KUKA KRL program: MyProgram_014().src

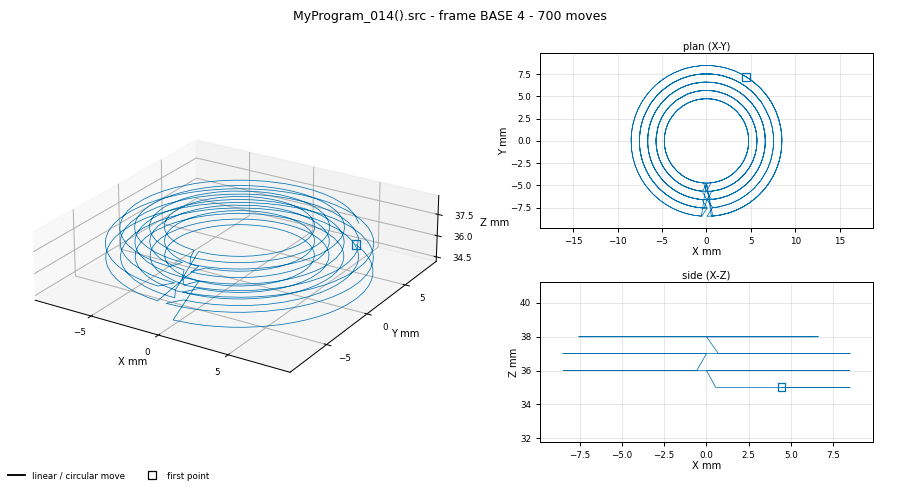
[picture p0: tool path of MyProgram_014().src in frame BASE 4, 700 of 700 moves have a stored position in this frame; points joined in program order, loops and branches not executed]
&ACCESS RVP
&REL 1
&PARAM TEMPLATE = C:\KRC\Roboter\Template\vorgabe
&PARAM EDITMASK = *
DEF MyProgram_014()
; ---- Setting reference (Base) ----
$BASE = BASE_DATA[4]

; --------------------------
; ---- Setting tool (TCP) ----
$TOOL = TOOL_DATA[3]
; --------------------------

$VEL.CP = VEL_APROX_PRINT
Startdeposition()
$VEL.CP = VEL_PRINT
LIN {X 4.4354,Y 7.2394,Z 35,A -2.2302,B 0,C 0,E1 0.1598,E2 90.0725} C_DIS
LIN {X 5.4049,Y 6.549,Z 35,A -2.2236,B 0,C 0,E1 0.1598,E2 90.0723} C_DIS
LIN {X 6.1861,Y 5.8118,Z 35,A -2.2262,B 0,C 0,E1 0.1598,E2 90.0723} C_DIS
LIN {X 6.7419,Y 5.1563,Z 35,A -2.2336,B 0,C 0,E1 0.1598,E2 90.0723} C_DIS
LIN {X 7.2287,Y 4.4482,Z 35,A -2.2457,B 0,C 0,E1 0.1598,E2 90.0723} C_DIS
LIN {X 7.6414,Y 3.6945,Z 35,A -2.2626,B 0,C 0,E1 0.1598,E2 90.0723} C_DIS
LIN {X 7.9758,Y 2.9029,Z 35,A -2.2839,B 0,C 0,E1 0.1598,E2 90.0721} C_DIS
LIN {X 8.2282,Y 2.0814,Z 35,A -2.3096,B 0,C 0,E1 0.1598,E2 90.0721} C_DIS
LIN {X 8.3959,Y 1.2387,Z 35,A -2.3393,B 0,C 0,E1 0.1598,E2 90.0721} C_DIS
LIN {X 8.4889,Y 0.1686,Z 35,A -2.3812,B 0,C 0,E1 0.1598,E2 90.0716} C_DIS
LIN {X 8.427,Y -1.0082,Z 35,A -2.4336,B 0,C 0,E1 0.1598,E2 90.0716} C_DIS
LIN {X 8.2841,Y -1.8426,Z 35,A -2.4748,B 0,C 0,E1 0.1598,E2 90.0719} C_DIS
LIN {X 8.0591,Y -2.6586,Z 35,A -2.5179,B 0,C 0,E1 0.1598,E2 90.0719} C_DIS
LIN {X 7.754,Y -3.4482,Z 35,A -2.5628,B 0,C 0,E1 0.1598,E2 90.0719} C_DIS
LIN {X 7.3718,Y -4.2035,Z 35,A -2.6091,B 0,C 0,E1 0.1598,E2 90.0718} C_DIS
LIN {X 6.9163,Y -4.9169,Z 35,A -2.6563,B 0,C 0,E1 0.1598,E2 90.0718} C_DIS
LIN {X 6.3921,Y -5.5815,Z 35,A -2.7039,B 0,C 0,E1 0.1598,E2 90.0718} C_DIS
LIN {X 5.5803,Y -6.3989,Z 35,A -2.7685,B 0,C 0,E1 0.1598,E2 90.0716} C_DIS
LIN {X 4.7589,Y -7.0287,Z 35,A -2.8256,B 0,C 0,E1 0.1598,E2 90.0716} C_DIS
LIN {X 4.0513,Y -7.4589,Z 35,A -2.8699,B 0,C 0,E1 0.1598,E2 90.0716} C_DIS
LIN {X 3.3051,Y -7.8178,Z 35,A -2.9126,B 0,C 0,E1 0.1598,E2 90.0716} C_DIS
LIN {X 2.5274,Y -8.1021,Z 35,A -2.9533,B 0,C 0,E1 0.1598,E2 90.0716} C_DIS
LIN {X 1.7257,Y -8.3091,Z 35,A -2.9915,B 0,C 0,E1 0.1598,E2 90.0716} C_DIS
LIN {X 0.5478,Y -8.4729,Z 35,A -3.0416,B 0,C 0,E1 0.1598,E2 90.0716} C_DIS
LIN {X 0.5478,Y -8.4729,Z 35,A -3.0416,B 0,C 0,E1 0.1598,E2 90.0716} C_DIS
Enddeposition()
LIN {X 0.0007,Y -4.7534,Z 36,A -2.8887,B 0,C 0,E1 0.1598,E2 90.0604} C_DIS
Startdeposition()
$VEL.CP = VEL_PRINT
LIN {X 0.0007,Y -4.7534,Z 36,A -2.8945,B 0,C 0,E1 0.1598,E2 90.0661} C_DIS
LIN {X 0.8257,Y -4.6787,Z 36,A -2.8659,B 0,C 0,E1 0.1598,E2 90.0711} C_DIS
LIN {X 1.4687,Y -4.5179,Z 36,A -2.8361,B 0,C 0,E1 0.1598,E2 90.0717} C_DIS
LIN {X 2.0836,Y -4.2702,Z 36,A -2.803,B 0,C 0,E1 0.1598,E2 90.0718} C_DIS
LIN {X 2.6574,Y -3.9383,Z 36,A -2.7678,B 0,C 0,E1 0.1598,E2 90.0718} C_DIS
LIN {X 3.2997,Y -3.4155,Z 36,A -2.7219,B 0,C 0,E1 0.1598,E2 90.0718} C_DIS
LIN {X 3.7426,Y -2.9228,Z 36,A -2.6846,B 0,C 0,E1 0.1598,E2 90.0718} C_DIS
LIN {X 4.1951,Y -2.2293,Z 36,A -2.6384,B 0,C 0,E1 0.1598,E2 90.0718} C_DIS
LIN {X 4.4644,Y -1.6239,Z 36,A -2.6027,B 0,C 0,E1 0.1598,E2 90.0719} C_DIS
LIN {X 4.6471,Y -0.9868,Z 36,A -2.5689,B 0,C 0,E1 0.1598,E2 90.0719} C_DIS
LIN {X 4.7402,Y -0.3306,Z 36,A -2.5375,B 0,C 0,E1 0.1598,E2 90.0719} C_DIS
LIN {X 4.74,Y 0.3322,Z 36,A -2.5093,B 0,C 0,E1 0.1598,E2 90.0719} C_DIS
LIN {X 4.6474,Y 0.9886,Z 36,A -2.4848,B 0,C 0,E1 0.1598,E2 90.072} C_DIS
LIN {X 4.4647,Y 1.6257,Z 36,A -2.4644,B 0,C 0,E1 0.1598,E2 90.072} C_DIS
LIN {X 4.1961,Y 2.2319,Z 36,A -2.4485,B 0,C 0,E1 0.1598,E2 90.072} C_DIS
LIN {X 3.8438,Y 2.7936,Z 36,A -2.4376,B 0,C 0,E1 0.1598,E2 90.0721} C_DIS
LIN {X 3.4175,Y 3.3013,Z 36,A -2.4318,B 0,C 0,E1 0.1598,E2 90.0721} C_DIS
LIN {X 2.9251,Y 3.7453,Z 36,A -2.4311,B 0,C 0,E1 0.1598,E2 90.0722} C_DIS
LIN {X 2.3754,Y 4.116,Z 36,A -2.4357,B 0,C 0,E1 0.1598,E2 90.0722} C_DIS
LIN {X 1.7795,Y 4.4064,Z 36,A -2.4453,B 0,C 0,E1 0.1598,E2 90.0722} C_DIS
LIN {X 1.149,Y 4.6114,Z 36,A -2.4599,B 0,C 0,E1 0.1598,E2 90.0722} C_DIS
LIN {X 0.4961,Y 4.7268,Z 36,A -2.4791,B 0,C 0,E1 0.1598,E2 90.0722} C_DIS
LIN {X -0.1665,Y 4.7482,Z 36,A -2.5026,B 0,C 0,E1 0.1598,E2 90.0722} C_DIS
LIN {X -0.8256,Y 4.6784,Z 36,A -2.5299,B 0,C 0,E1 0.1598,E2 90.0722} C_DIS
LIN {X -1.4684,Y 4.5172,Z 36,A -2.5604,B 0,C 0,E1 0.1598,E2 90.0722} C_DIS
LIN {X -2.083,Y 4.269,Z 36,A -2.5935,B 0,C 0,E1 0.1598,E2 90.0721} C_DIS
LIN {X -2.6569,Y 3.9376,Z 36,A -2.6287,B 0,C 0,E1 0.1598,E2 90.0721} C_DIS
LIN {X -3.1791,Y 3.5295,Z 36,A -2.6652,B 0,C 0,E1 0.1598,E2 90.0719} C_DIS
LIN {X -3.6394,Y 3.0527,Z 36,A -2.7023,B 0,C 0,E1 0.1598,E2 90.0719} C_DIS
LIN {X -4.0291,Y 2.5166,Z 36,A -2.7393,B 0,C 0,E1 0.1598,E2 90.0718} C_DIS
LIN {X -4.342,Y 1.9322,Z 36,A -2.7755,B 0,C 0,E1 0.1598,E2 90.0717} C_DIS
LIN {X -4.5683,Y 1.3091,Z 36,A -2.8102,B 0,C 0,E1 0.1598,E2 90.0717} C_DIS
LIN {X -4.7045,Y 0.6604,Z 36,A -2.8426,B 0,C 0,E1 0.1598,E2 90.0716} C_DIS
LIN {X -4.7508,Y -0.0007,Z 36,A -2.8723,B 0,C 0,E1 0.1598,E2 90.0716} C_DIS
LIN {X -4.7064,Y -0.6622,Z 36,A -2.8987,B 0,C 0,E1 0.1598,E2 90.0715} C_DIS
LIN {X -4.5654,Y -1.3099,Z 36,A -2.9209,B 0,C 0,E1 0.1598,E2 90.0715} C_DIS
LIN {X -4.3396,Y -1.9329,Z 36,A -2.939,B 0,C 0,E1 0.1598,E2 90.0715} C_DIS
LIN {X -4.0299,Y -2.519,Z 36,A -2.9525,B 0,C 0,E1 0.1598,E2 90.0715} C_DIS
LIN {X -3.6397,Y -3.0551,Z 36,A -2.9609,B 0,C 0,E1 0.1598,E2 90.0715} C_DIS
LIN {X -3.1791,Y -3.532,Z 36,A -2.9643,B 0,C 0,E1 0.1598,E2 90.0715} C_DIS
LIN {X -2.6569,Y -3.9405,Z 36,A -2.9624,B 0,C 0,E1 0.1598,E2 90.0715} C_DIS
LIN {X -2.0828,Y -4.2724,Z 36,A -2.9555,B 0,C 0,E1 0.1598,E2 90.0715} C_DIS
LIN {X -1.4676,Y -4.5196,Z 36,A -2.9434,B 0,C 0,E1 0.1598,E2 90.0716} C_DIS
LIN {X -0.8243,Y -4.6796,Z 36,A -2.9266,B 0,C 0,E1 0.1598,E2 90.0716} C_DIS
LIN {X 0.0007,Y -4.7534,Z 36,A -2.8995,B 0,C 0,E1 0.1598,E2 90.0717} C_DIS
Enddeposition()
LIN {X 0.0007,Y -4.7534,Z 36,A -2.8995,B 0,C 0,E1 0.1598,E2 90.0717} C_DIS
Startdeposition()
$VEL.CP = VEL_PRINT
LIN {X -0.4227,Y -5.6705,Z 36,A -2.9535,B 0,C 0,E1 0.1598,E2 90.0711} C_DIS
LIN {X -1.1482,Y -5.5725,Z 36,A -2.9765,B 0,C 0,E1 0.1598,E2 90.0716} C_DIS
LIN {X -2.3524,Y -5.18,Z 36,A -3.004,B 0,C 0,E1 0.1598,E2 90.0715} C_DIS
LIN {X -3.1624,Y -4.7301,Z 36,A -3.0146,B 0,C 0,E1 0.1598,E2 90.0715} C_DIS
LIN {X -3.9702,Y -4.069,Z 36,A -3.0161,B 0,C 0,E1 0.1598,E2 90.0713} C_DIS
LIN {X -4.5224,Y -3.4424,Z 36,A -3.0098,B 0,C 0,E1 0.1598,E2 90.0713} C_DIS
LIN {X -4.9778,Y -2.7426,Z 36,A -2.9969,B 0,C 0,E1 0.1598,E2 90.0713} C_DIS
LIN {X -5.3253,Y -1.9835,Z 36,A -2.9774,B 0,C 0,E1 0.1598,E2 90.0713} C_DIS
LIN {X -5.5586,Y -1.1818,Z 36,A -2.952,B 0,C 0,E1 0.1598,E2 90.0713} C_DIS
LIN {X -5.672,Y -0.3547,Z 36,A -2.9212,B 0,C 0,E1 0.1598,E2 90.0713} C_DIS
LIN {X -5.6631,Y 0.4802,Z 36,A -2.8855,B 0,C 0,E1 0.1598,E2 90.0713} C_DIS
LIN {X -5.5325,Y 1.3049,Z 36,A -2.8458,B 0,C 0,E1 0.1598,E2 90.0714} C_DIS
LIN {X -5.2826,Y 2.1019,Z 36,A -2.8029,B 0,C 0,E1 0.1598,E2 90.0715} C_DIS
LIN {X -4.9174,Y 2.853,Z 36,A -2.7578,B 0,C 0,E1 0.1598,E2 90.0716} C_DIS
LIN {X -4.4466,Y 3.543,Z 36,A -2.7113,B 0,C 0,E1 0.1598,E2 90.0717} C_DIS
LIN {X -3.8784,Y 4.1552,Z 36,A -2.6645,B 0,C 0,E1 0.1598,E2 90.0718} C_DIS
LIN {X -3.2282,Y 4.6792,Z 36,A -2.6184,B 0,C 0,E1 0.1598,E2 90.0719} C_DIS
LIN {X -2.5072,Y 5.1007,Z 36,A -2.574,B 0,C 0,E1 0.1598,E2 90.0721} C_DIS
LIN {X -1.7329,Y 5.4131,Z 36,A -2.5323,B 0,C 0,E1 0.1598,E2 90.0721} C_DIS
LIN {X -0.9211,Y 5.6088,Z 36,A -2.4941,B 0,C 0,E1 0.1598,E2 90.0722} C_DIS
LIN {X -0.0893,Y 5.6818,Z 36,A -2.4603,B 0,C 0,E1 0.1598,E2 90.0722} C_DIS
LIN {X 0.744,Y 5.6331,Z 36,A -2.4317,B 0,C 0,E1 0.1598,E2 90.0723} C_DIS
LIN {X 1.5615,Y 5.4639,Z 36,A -2.4087,B 0,C 0,E1 0.1598,E2 90.0723} C_DIS
LIN {X 2.3448,Y 5.1756,Z 36,A -2.392,B 0,C 0,E1 0.1598,E2 90.0723} C_DIS
LIN {X 3.0781,Y 4.7766,Z 36,A -2.3818,B 0,C 0,E1 0.1598,E2 90.0723} C_DIS
LIN {X 3.7445,Y 4.2737,Z 36,A -2.3786,B 0,C 0,E1 0.1598,E2 90.0723} C_DIS
LIN {X 4.3303,Y 3.6789,Z 36,A -2.3822,B 0,C 0,E1 0.1598,E2 90.0722} C_DIS
LIN {X 4.8227,Y 3.0048,Z 36,A -2.3927,B 0,C 0,E1 0.1598,E2 90.0722} C_DIS
LIN {X 5.2114,Y 2.266,Z 36,A -2.4098,B 0,C 0,E1 0.1598,E2 90.072} C_DIS
LIN {X 5.5672,Y 1.1736,Z 36,A -2.4428,B 0,C 0,E1 0.1598,E2 90.0717} C_DIS
LIN {X 5.6752,Y 0.4058,Z 36,A -2.4718,B 0,C 0,E1 0.1598,E2 90.0719} C_DIS
LIN {X 5.6485,Y -0.684,Z 36,A -2.5189,B 0,C 0,E1 0.1598,E2 90.0715} C_DIS
LIN {X 5.464,Y -1.5648,Z 36,A -2.5634,B 0,C 0,E1 0.1598,E2 90.0717} C_DIS
LIN {X 5.2237,Y -2.2434,Z 36,A -2.6013,B 0,C 0,E1 0.1598,E2 90.0718} C_DIS
LIN {X 4.8083,Y -3.0416,Z 36,A -2.6504,B 0,C 0,E1 0.1598,E2 90.0717} C_DIS
LIN {X 4.0645,Y -3.9725,Z 36,A -2.7174,B 0,C 0,E1 0.1598,E2 90.0715} C_DIS
LIN {X 3.4798,Y -4.495,Z 36,A -2.7613,B 0,C 0,E1 0.1598,E2 90.0717} C_DIS
LIN {X 2.8282,Y -4.9317,Z 36,A -2.8039,B 0,C 0,E1 0.1598,E2 90.0717} C_DIS
LIN {X 2.1227,Y -5.2744,Z 36,A -2.8444,B 0,C 0,E1 0.1598,E2 90.0717} C_DIS
LIN {X 1.3766,Y -5.5169,Z 36,A -2.8821,B 0,C 0,E1 0.1598,E2 90.0717} C_DIS
LIN {X 0.6041,Y -5.6533,Z 36,A -2.9163,B 0,C 0,E1 0.1598,E2 90.0717} C_DIS
LIN {X 0.6041,Y -5.6533,Z 36,A -2.9163,B 0,C 0,E1 0.1598,E2 90.0717} C_DIS
Enddeposition()
LIN {X 0.0318,Y -6.6195,Z 36,A -2.9773,B 0,C 0,E1 0.1598,E2 90.0704} C_DIS
Startdeposition()
$VEL.CP = VEL_PRINT
LIN {X 0.9472,Y -6.552,Z 36,A -2.942,B 0,C 0,E1 0.1598,E2 90.0716} C_DIS
LIN {X 1.6671,Y -6.4068,Z 36,A -2.9095,B 0,C 0,E1 0.1598,E2 90.0716} C_DIS
LIN {X 2.3666,Y -6.1835,Z 36,A -2.8743,B 0,C 0,E1 0.1598,E2 90.0717} C_DIS
LIN {X 3.036,Y -5.8815,Z 36,A -2.8369,B 0,C 0,E1 0.1598,E2 90.0717} C_DIS
LIN {X 3.6694,Y -5.5096,Z 36,A -2.7978,B 0,C 0,E1 0.1598,E2 90.0717} C_DIS
LIN {X 4.258,Y -5.0704,Z 36,A -2.7575,B 0,C 0,E1 0.1598,E2 90.0718} C_DIS
LIN {X 4.7941,Y -4.5683,Z 36,A -2.7164,B 0,C 0,E1 0.1598,E2 90.0718} C_DIS
LIN {X 5.269,Y -4.0081,Z 36,A -2.675,B 0,C 0,E1 0.1598,E2 90.0718} C_DIS
LIN {X 5.6805,Y -3.3996,Z 36,A -2.6339,B 0,C 0,E1 0.1598,E2 90.0718} C_DIS
LIN {X 6.022,Y -2.7493,Z 36,A -2.5936,B 0,C 0,E1 0.1598,E2 90.0718} C_DIS
LIN {X 6.2882,Y -2.0649,Z 36,A -2.5547,B 0,C 0,E1 0.1598,E2 90.0719} C_DIS
LIN {X 6.4796,Y -1.3558,Z 36,A -2.5174,B 0,C 0,E1 0.1598,E2 90.0719} C_DIS
LIN {X 6.589,Y -0.6295,Z 36,A -2.4824,B 0,C 0,E1 0.1598,E2 90.0719} C_DIS
LIN {X 6.6176,Y 0.1041,Z 36,A -2.4501,B 0,C 0,E1 0.1598,E2 90.0719} C_DIS
LIN {X 6.5658,Y 0.8366,Z 36,A -2.4208,B 0,C 0,E1 0.1598,E2 90.072} C_DIS
LIN {X 6.4327,Y 1.5587,Z 36,A -2.3949,B 0,C 0,E1 0.1598,E2 90.072} C_DIS
LIN {X 6.2216,Y 2.2623,Z 36,A -2.3727,B 0,C 0,E1 0.1598,E2 90.0721} C_DIS
LIN {X 5.9327,Y 2.9374,Z 36,A -2.3547,B 0,C 0,E1 0.1598,E2 90.0721} C_DIS
LIN {X 5.5705,Y 3.5762,Z 36,A -2.3408,B 0,C 0,E1 0.1598,E2 90.0722} C_DIS
LIN {X 5.1397,Y 4.171,Z 36,A -2.3314,B 0,C 0,E1 0.1598,E2 90.0722} C_DIS
LIN {X 4.646,Y 4.7148,Z 36,A -2.3265,B 0,C 0,E1 0.1598,E2 90.0722} C_DIS
LIN {X 3.8364,Y 5.3992,Z 36,A -2.3272,B 0,C 0,E1 0.1598,E2 90.0722} C_DIS
LIN {X 3.0111,Y 5.895,Z 36,A -2.3367,B 0,C 0,E1 0.1598,E2 90.0723} C_DIS
LIN {X 2.3065,Y 6.2065,Z 36,A -2.3496,B 0,C 0,E1 0.1598,E2 90.0723} C_DIS
LIN {X 1.5698,Y 6.4311,Z 36,A -2.3672,B 0,C 0,E1 0.1598,E2 90.0723} C_DIS
LIN {X 0.4931,Y 6.6051,Z 36,A -2.3996,B 0,C 0,E1 0.1598,E2 90.0723} C_DIS
LIN {X -0.4931,Y 6.6051,Z 36,A -2.436,B 0,C 0,E1 0.1598,E2 90.0723} C_DIS
LIN {X -1.5396,Y 6.4379,Z 36,A -2.4817,B 0,C 0,E1 0.1598,E2 90.0723} C_DIS
LIN {X -2.2379,Y 6.228,Z 36,A -2.5163,B 0,C 0,E1 0.1598,E2 90.0722} C_DIS
LIN {X -2.9104,Y 5.946,Z 36,A -2.5531,B 0,C 0,E1 0.1598,E2 90.0722} C_DIS
LIN {X -3.5465,Y 5.5892,Z 36,A -2.5916,B 0,C 0,E1 0.1598,E2 90.0721} C_DIS
LIN {X -4.1402,Y 5.1658,Z 36,A -2.6314,B 0,C 0,E1 0.1598,E2 90.072} C_DIS
LIN {X -4.6831,Y 4.6788,Z 36,A -2.6719,B 0,C 0,E1 0.1598,E2 90.0719} C_DIS
LIN {X -5.1686,Y 4.1348,Z 36,A -2.7128,B 0,C 0,E1 0.1598,E2 90.0719} C_DIS
LIN {X -5.5916,Y 3.5409,Z 36,A -2.7535,B 0,C 0,E1 0.1598,E2 90.0717} C_DIS
LIN {X -5.9473,Y 2.9044,Z 36,A -2.7934,B 0,C 0,E1 0.1598,E2 90.0717} C_DIS
LIN {X -6.2297,Y 2.2321,Z 36,A -2.8322,B 0,C 0,E1 0.1598,E2 90.0716} C_DIS
LIN {X -6.4395,Y 1.5339,Z 36,A -2.8695,B 0,C 0,E1 0.1598,E2 90.0715} C_DIS
LIN {X -6.6051,Y 0.4931,Z 36,A -2.9193,B 0,C 0,E1 0.1598,E2 90.0711} C_DIS
LIN {X -6.6084,Y -0.4169,Z 36,A -2.958,B 0,C 0,E1 0.1598,E2 90.0712} C_DIS
LIN {X -6.5197,Y -1.1393,Z 36,A -2.9854,B 0,C 0,E1 0.1598,E2 90.0713} C_DIS
LIN {X -6.3558,Y -1.8484,Z 36,A -3.0094,B 0,C 0,E1 0.1598,E2 90.0713} C_DIS
LIN {X -6.1157,Y -2.5355,Z 36,A -3.0297,B 0,C 0,E1 0.1598,E2 90.0713} C_DIS
LIN {X -5.8012,Y -3.1919,Z 36,A -3.0459,B 0,C 0,E1 0.1598,E2 90.0713} C_DIS
LIN {X -5.4138,Y -3.8082,Z 36,A -3.0578,B 0,C 0,E1 0.1598,E2 90.0713} C_DIS
LIN {X -4.9632,Y -4.3798,Z 36,A -3.0655,B 0,C 0,E1 0.1598,E2 90.0713} C_DIS
LIN {X -4.4519,Y -4.898,Z 36,A -3.0687,B 0,C 0,E1 0.1598,E2 90.0713} C_DIS
LIN {X -3.8874,Y -5.3575,Z 36,A -3.0675,B 0,C 0,E1 0.1598,E2 90.0713} C_DIS
LIN {X -3.2766,Y -5.7531,Z 36,A -3.0619,B 0,C 0,E1 0.1598,E2 90.0714} C_DIS
LIN {X -2.6243,Y -6.0759,Z 36,A -3.0517,B 0,C 0,E1 0.1598,E2 90.0714} C_DIS
LIN {X -1.9411,Y -6.3265,Z 36,A -3.0373,B 0,C 0,E1 0.1598,E2 90.0714} C_DIS
LIN {X -1.2354,Y -6.5045,Z 36,A -3.019,B 0,C 0,E1 0.1598,E2 90.0715} C_DIS
LIN {X -0.5139,Y -6.5993,Z 36,A -2.9966,B 0,C 0,E1 0.1598,E2 90.0715} C_DIS
LIN {X -0.5139,Y -6.5993,Z 36,A -2.9966,B 0,C 0,E1 0.1598,E2 90.0715} C_DIS
Enddeposition()
LIN {X 0.0763,Y -7.5547,Z 36,A -3.0146,B 0,C 0,E1 0.1598,E2 90.0704} C_DIS
Startdeposition()
$VEL.CP = VEL_PRINT
LIN {X -0.5178,Y -7.5391,Z 36,A -3.0368,B 0,C 0,E1 0.1598,E2 90.0715} C_DIS
LIN {X -1.5892,Y -7.3847,Z 36,A -3.0696,B 0,C 0,E1 0.1598,E2 90.0715} C_DIS
LIN {X -2.4237,Y -7.153,Z 36,A -3.0903,B 0,C 0,E1 0.1598,E2 90.0715} C_DIS
LIN {X -3.5202,Y -6.6878,Z 36,A -3.1107,B 0,C 0,E1 0.1598,E2 90.0713} C_DIS
LIN {X -4.4245,Y -6.122,Z 36,A -3.1198,B 0,C 0,E1 0.1598,E2 90.0713} C_DIS
LIN {X -5.3543,Y -5.335,Z 36,A -3.1204,B 0,C 0,E1 0.1598,E2 90.0711} C_DIS
LIN {X -5.9738,Y -4.6194,Z 36,A -3.1129,B 0,C 0,E1 0.1598,E2 90.0711} C_DIS
LIN {X -6.4079,Y -3.999,Z 36,A -3.1026,B 0,C 0,E1 0.1598,E2 90.0712} C_DIS
LIN {X -6.776,Y -3.3373,Z 36,A -3.0881,B 0,C 0,E1 0.1598,E2 90.0712} C_DIS
LIN {X -7.0765,Y -2.6424,Z 36,A -3.0697,B 0,C 0,E1 0.1598,E2 90.0712} C_DIS
LIN {X -7.3059,Y -1.9207,Z 36,A -3.0476,B 0,C 0,E1 0.1598,E2 90.0712} C_DIS
LIN {X -7.4927,Y -0.9928,Z 36,A -3.0149,B 0,C 0,E1 0.1598,E2 90.071} C_DIS
LIN {X -7.5499,Y 0.2371,Z 36,A -2.9648,B 0,C 0,E1 0.1598,E2 90.0708} C_DIS
LIN {X -7.417,Y 1.45,Z 36,A -2.9087,B 0,C 0,E1 0.1598,E2 90.0709} C_DIS
LIN {X -7.1726,Y 2.3819,Z 36,A -2.8606,B 0,C 0,E1 0.1598,E2 90.0713} C_DIS
LIN {X -6.7301,Y 3.4283,Z 36,A -2.7999,B 0,C 0,E1 0.1598,E2 90.0713} C_DIS
LIN {X -6.2262,Y 4.2818,Z 36,A -2.7454,B 0,C 0,E1 0.1598,E2 90.0715} C_DIS
LIN {X -5.5374,Y 5.1423,Z 36,A -2.6837,B 0,C 0,E1 0.1598,E2 90.0716} C_DIS
LIN {X -4.9739,Y 5.6849,Z 36,A -2.6403,B 0,C 0,E1 0.1598,E2 90.0719} C_DIS
LIN {X -4.0486,Y 6.381,Z 36,A -2.5766,B 0,C 0,E1 0.1598,E2 90.0719} C_DIS
LIN {X -2.7827,Y 7.0219,Z 36,A -2.5028,B 0,C 0,E1 0.1598,E2 90.072} C_DIS
LIN {X -1.6837,Y 7.368,Z 36,A -2.4478,B 0,C 0,E1 0.1598,E2 90.0723} C_DIS
LIN {X -0.4157,Y 7.546,Z 36,A -2.3935,B 0,C 0,E1 0.1598,E2 90.0723} C_DIS
LIN {X 1.1377,Y 7.4709,Z 36,A -2.3393,B 0,C 0,E1 0.1598,E2 90.0724} C_DIS
LIN {X 2.0218,Y 7.2822,Z 36,A -2.3146,B 0,C 0,E1 0.1598,E2 90.0724} C_DIS
LIN {X 3.3395,Y 6.7787,Z 36,A -2.2873,B 0,C 0,E1 0.1598,E2 90.0724} C_DIS
LIN {X 4.2884,Y 6.216,Z 36,A -2.2761,B 0,C 0,E1 0.1598,E2 90.0724} C_DIS
LIN {X 4.8709,Y 5.7707,Z 36,A -2.2736,B 0,C 0,E1 0.1598,E2 90.0724} C_DIS
LIN {X 5.4093,Y 5.2728,Z 36,A -2.2749,B 0,C 0,E1 0.1598,E2 90.0724} C_DIS
LIN {X 6.1007,Y 4.4625,Z 36,A -2.2837,B 0,C 0,E1 0.1598,E2 90.0721} C_DIS
LIN {X 6.6299,Y 3.6229,Z 36,A -2.2999,B 0,C 0,E1 0.1598,E2 90.0721} C_DIS
LIN {X 7.0498,Y 2.7236,Z 36,A -2.3225,B 0,C 0,E1 0.1598,E2 90.0719} C_DIS
LIN {X 7.4177,Y 1.4467,Z 36,A -2.363,B 0,C 0,E1 0.1598,E2 90.0715} C_DIS
LIN {X 7.5393,Y 0.5152,Z 36,A -2.3986,B 0,C 0,E1 0.1598,E2 90.0719} C_DIS
LIN {X 7.5255,Y -0.6346,Z 36,A -2.4479,B 0,C 0,E1 0.1598,E2 90.0716} C_DIS
LIN {X 7.4171,Y -1.4177,Z 36,A -2.4857,B 0,C 0,E1 0.1598,E2 90.0719} C_DIS
LIN {X 7.2299,Y -2.1858,Z 36,A -2.5253,B 0,C 0,E1 0.1598,E2 90.0719} C_DIS
LIN {X 6.9601,Y -2.9289,Z 36,A -2.5669,B 0,C 0,E1 0.1598,E2 90.0719} C_DIS
LIN {X 6.6176,Y -3.6415,Z 36,A -2.6099,B 0,C 0,E1 0.1598,E2 90.0719} C_DIS
LIN {X 6.0082,Y -4.5828,Z 36,A -2.6723,B 0,C 0,E1 0.1598,E2 90.0716} C_DIS
LIN {X 5.3287,Y -5.3604,Z 36,A -2.7304,B 0,C 0,E1 0.1598,E2 90.0716} C_DIS
LIN {X 4.539,Y -6.0374,Z 36,A -2.7884,B 0,C 0,E1 0.1598,E2 90.0716} C_DIS
LIN {X 3.6683,Y -6.6064,Z 36,A -2.8446,B 0,C 0,E1 0.1598,E2 90.0716} C_DIS
LIN {X 2.6344,Y -7.081,Z 36,A -2.9028,B 0,C 0,E1 0.1598,E2 90.0716} C_DIS
LIN {X 1.5886,Y -7.388,Z 36,A -2.9543,B 0,C 0,E1 0.1598,E2 90.0716} C_DIS
LIN {X 0.6836,Y -7.5258,Z 36,A -2.9934,B 0,C 0,E1 0.1598,E2 90.0716} C_DIS
LIN {X 0.6836,Y -7.5258,Z 36,A -2.9934,B 0,C 0,E1 0.1598,E2 90.0716} C_DIS
Enddeposition()
LIN {X 0.061,Y -8.4892,Z 36,A -3.0562,B 0,C 0,E1 0.1598,E2 90.0703} C_DIS
Startdeposition()
$VEL.CP = VEL_PRINT
LIN {X 1.059,Y -8.4194,Z 36,A -3.0178,B 0,C 0,E1 0.1598,E2 90.0715} C_DIS
LIN {X 1.8475,Y -8.2823,Z 36,A -2.9831,B 0,C 0,E1 0.1598,E2 90.0715} C_DIS
LIN {X 2.6197,Y -8.0718,Z 36,A -2.9458,B 0,C 0,E1 0.1598,E2 90.0716} C_DIS
LIN {X 3.3687,Y -7.7897,Z 36,A -2.9063,B 0,C 0,E1 0.1598,E2 90.0716} C_DIS
LIN {X 4.0879,Y -7.4383,Z 36,A -2.865,B 0,C 0,E1 0.1598,E2 90.0716} C_DIS
LIN {X 4.7707,Y -7.0205,Z 36,A -2.8221,B 0,C 0,E1 0.1598,E2 90.0717} C_DIS
LIN {X 5.7221,Y -6.2743,Z 36,A -2.7552,B 0,C 0,E1 0.1598,E2 90.0717} C_DIS
LIN {X 6.5818,Y -5.3568,Z 36,A -2.6843,B 0,C 0,E1 0.1598,E2 90.0715} C_DIS
LIN {X 7.0892,Y -4.6648,Z 36,A -2.6364,B 0,C 0,E1 0.1598,E2 90.0718} C_DIS
LIN {X 7.5242,Y -3.9252,Z 36,A -2.5888,B 0,C 0,E1 0.1598,E2 90.0718} C_DIS
LIN {X 7.8824,Y -3.1453,Z 36,A -2.5424,B 0,C 0,E1 0.1598,E2 90.0718} C_DIS
LIN {X 8.16,Y -2.3334,Z 36,A -2.4975,B 0,C 0,E1 0.1598,E2 90.0718} C_DIS
LIN {X 8.3544,Y -1.4975,Z 36,A -2.4546,B 0,C 0,E1 0.1598,E2 90.0719} C_DIS
LIN {X 8.4639,Y -0.6464,Z 36,A -2.4143,B 0,C 0,E1 0.1598,E2 90.0719} C_DIS
LIN {X 8.4734,Y 0.5391,Z 36,A -2.363,B 0,C 0,E1 0.1598,E2 90.0717} C_DIS
LIN {X 8.3331,Y 1.6129,Z 36,A -2.3225,B 0,C 0,E1 0.1598,E2 90.0719} C_DIS
LIN {X 8.1256,Y 2.4541,Z 36,A -2.2945,B 0,C 0,E1 0.1598,E2 90.0721} C_DIS
LIN {X 7.8332,Y 3.2697,Z 36,A -2.2705,B 0,C 0,E1 0.1598,E2 90.0721} C_DIS
LIN {X 7.4589,Y 4.0511,Z 36,A -2.2511,B 0,C 0,E1 0.1598,E2 90.0722} C_DIS
LIN {X 7.007,Y 4.7902,Z 36,A -2.2363,B 0,C 0,E1 0.1598,E2 90.0722} C_DIS
LIN {X 6.4821,Y 5.4796,Z 36,A -2.2264,B 0,C 0,E1 0.1598,E2 90.0723} C_DIS
LIN {X 5.89,Y 6.1121,Z 36,A -2.2213,B 0,C 0,E1 0.1598,E2 90.0723} C_DIS
LIN {X 4.8948,Y 6.9375,Z 36,A -2.2228,B 0,C 0,E1 0.1598,E2 90.0722} C_DIS
LIN {X 3.8666,Y 7.5552,Z 36,A -2.2346,B 0,C 0,E1 0.1598,E2 90.0723} C_DIS
LIN {X 3.0744,Y 7.9105,Z 36,A -2.249,B 0,C 0,E1 0.1598,E2 90.0725} C_DIS
LIN {X 2.2502,Y 8.1832,Z 36,A -2.2679,B 0,C 0,E1 0.1598,E2 90.0725} C_DIS
LIN {X 1.4026,Y 8.3708,Z 36,A -2.2912,B 0,C 0,E1 0.1598,E2 90.0725} C_DIS
LIN {X 0.5403,Y 8.471,Z 36,A -2.3188,B 0,C 0,E1 0.1598,E2 90.0725} C_DIS
LIN {X -0.7485,Y 8.4591,Z 36,A -2.367,B 0,C 0,E1 0.1598,E2 90.0725} C_DIS
LIN {X -2.004,Y 8.2471,Z 36,A -2.4223,B 0,C 0,E1 0.1598,E2 90.0723} C_DIS
LIN {X -2.7754,Y 8.0254,Z 36,A -2.4601,B 0,C 0,E1 0.1598,E2 90.0723} C_DIS
LIN {X -3.7432,Y 7.6164,Z 36,A -2.5131,B 0,C 0,E1 0.1598,E2 90.0722} C_DIS
LIN {X -4.4785,Y 7.2088,Z 36,A -2.5575,B 0,C 0,E1 0.1598,E2 90.0721} C_DIS
LIN {X -5.1698,Y 6.7305,Z 36,A -2.6031,B 0,C 0,E1 0.1598,E2 90.072} C_DIS
LIN {X -5.8108,Y 6.1865,Z 36,A -2.6497,B 0,C 0,E1 0.1598,E2 90.0719} C_DIS
LIN {X -6.5986,Y 5.3456,Z 36,A -2.7141,B 0,C 0,E1 0.1598,E2 90.0716} C_DIS
LIN {X -7.2974,Y 4.3327,Z 36,A -2.7824,B 0,C 0,E1 0.1598,E2 90.0713} C_DIS
LIN {X -7.7064,Y 3.5549,Z 36,A -2.8306,B 0,C 0,E1 0.1598,E2 90.0715} C_DIS
LIN {X -8.0327,Y 2.739,Z 36,A -2.877,B 0,C 0,E1 0.1598,E2 90.0714} C_DIS
LIN {X -8.338,Y 1.6073,Z 36,A -2.9358,B 0,C 0,E1 0.1598,E2 90.0711} C_DIS
LIN {X -8.4765,Y 0.4201,Z 36,A -2.991,B 0,C 0,E1 0.1598,E2 90.0709} C_DIS
LIN {X -8.4471,Y -0.8623,Z 36,A -3.0439,B 0,C 0,E1 0.1598,E2 90.0707} C_DIS
LIN {X -8.2625,Y -1.9348,Z 36,A -3.0827,B 0,C 0,E1 0.1598,E2 90.0709} C_DIS
LIN {X -8.0215,Y -2.7713,Z 36,A -3.1094,B 0,C 0,E1 0.1598,E2 90.0711} C_DIS
LIN {X -7.6957,Y -3.5787,Z 36,A -3.1316,B 0,C 0,E1 0.1598,E2 90.0711} C_DIS
LIN {X -7.2888,Y -4.3484,Z 36,A -3.1492,B 0,C 0,E1 0.1598,E2 90.0711} C_DIS
LIN {X -6.805,Y -5.0722,Z 36,A -3.1621,B 0,C 0,E1 0.1598,E2 90.0711} C_DIS
LIN {X -6.1023,Y -5.9032,Z 36,A -3.1714,B 0,C 0,E1 0.1598,E2 90.0709} C_DIS
LIN {X -5.2501,Y -6.6669,Z 36,A -3.1726,B 0,C 0,E1 0.1598,E2 90.0709} C_DIS
LIN {X -4.5591,Y -7.1572,Z 36,A -3.1682,B 0,C 0,E1 0.1598,E2 90.0712} C_DIS
LIN {X -3.8226,Y -7.5763,Z 36,A -3.1591,B 0,C 0,E1 0.1598,E2 90.0712} C_DIS
LIN {X -3.0481,Y -7.9199,Z 36,A -3.1453,B 0,C 0,E1 0.1598,E2 90.0713} C_DIS
LIN {X -2.2431,Y -8.1846,Z 36,A -3.1271,B 0,C 0,E1 0.1598,E2 90.0713} C_DIS
LIN {X -1.4158,Y -8.3678,Z 36,A -3.1045,B 0,C 0,E1 0.1598,E2 90.0714} C_DIS
LIN {X -0.5744,Y -8.4679,Z 36,A -3.078,B 0,C 0,E1 0.1598,E2 90.0714} C_DIS
LIN {X -0.5744,Y -8.4679,Z 36,A -3.078,B 0,C 0,E1 0.1598,E2 90.0714} C_DIS
Enddeposition()
LIN {X 0.0009,Y -4.7564,Z 37,A -2.8843,B 0,C 0,E1 0.1598,E2 90.0604} C_DIS
Startdeposition()
$VEL.CP = VEL_PRINT
LIN {X 0.0009,Y -4.7564,Z 37,A -2.89,B 0,C 0,E1 0.1598,E2 90.0661} C_DIS
LIN {X -0.8238,Y -4.6773,Z 37,A -2.9219,B 0,C 0,E1 0.1598,E2 90.071} C_DIS
LIN {X -1.4673,Y -4.519,Z 37,A -2.9394,B 0,C 0,E1 0.1598,E2 90.0716} C_DIS
LIN {X -2.082,Y -4.2709,Z 37,A -2.9514,B 0,C 0,E1 0.1598,E2 90.0716} C_DIS
LIN {X -2.6555,Y -3.9386,Z 37,A -2.9583,B 0,C 0,E1 0.1598,E2 90.0716} C_DIS
LIN {X -3.1779,Y -3.5307,Z 37,A -2.9602,B 0,C 0,E1 0.1598,E2 90.0716} C_DIS
LIN {X -3.6906,Y -2.9897,Z 37,A -2.956,B 0,C 0,E1 0.1598,E2 90.0715} C_DIS
LIN {X -4.0289,Y -2.5184,Z 37,A -2.9485,B 0,C 0,E1 0.1598,E2 90.0715} C_DIS
LIN {X -4.3395,Y -1.9329,Z 37,A -2.935,B 0,C 0,E1 0.1598,E2 90.0715} C_DIS
LIN {X -4.5665,Y -1.3101,Z 37,A -2.917,B 0,C 0,E1 0.1598,E2 90.0715} C_DIS
LIN {X -4.7045,Y -0.6619,Z 37,A -2.8946,B 0,C 0,E1 0.1598,E2 90.0715} C_DIS
LIN {X -4.7505,Y -0.0008,Z 37,A -2.8683,B 0,C 0,E1 0.1598,E2 90.0715} C_DIS
LIN {X -4.7058,Y 0.6605,Z 37,A -2.8386,B 0,C 0,E1 0.1598,E2 90.0715} C_DIS
LIN {X -4.5677,Y 1.3089,Z 37,A -2.8061,B 0,C 0,E1 0.1598,E2 90.0716} C_DIS
LIN {X -4.3407,Y 1.9316,Z 37,A -2.7714,B 0,C 0,E1 0.1598,E2 90.0716} C_DIS
LIN {X -4.0307,Y 2.5175,Z 37,A -2.7352,B 0,C 0,E1 0.1598,E2 90.0717} C_DIS
LIN {X -3.6407,Y 3.0537,Z 37,A -2.6982,B 0,C 0,E1 0.1598,E2 90.0718} C_DIS
LIN {X -3.1805,Y 3.531,Z 37,A -2.661,B 0,C 0,E1 0.1598,E2 90.0719} C_DIS
LIN {X -2.6584,Y 3.9396,Z 37,A -2.6245,B 0,C 0,E1 0.1598,E2 90.0719} C_DIS
LIN {X -2.0843,Y 4.2715,Z 37,A -2.5893,B 0,C 0,E1 0.1598,E2 90.0721} C_DIS
LIN {X -1.4696,Y 4.52,Z 37,A -2.5562,B 0,C 0,E1 0.1598,E2 90.0721} C_DIS
LIN {X -0.8261,Y 4.6789,Z 37,A -2.5257,B 0,C 0,E1 0.1598,E2 90.0721} C_DIS
LIN {X -0.1668,Y 4.749,Z 37,A -2.4985,B 0,C 0,E1 0.1598,E2 90.0722} C_DIS
LIN {X 0.4958,Y 4.7263,Z 37,A -2.475,B 0,C 0,E1 0.1598,E2 90.0722} C_DIS
LIN {X 1.1484,Y 4.6103,Z 37,A -2.4559,B 0,C 0,E1 0.1598,E2 90.0722} C_DIS
LIN {X 1.7786,Y 4.4051,Z 37,A -2.4413,B 0,C 0,E1 0.1598,E2 90.0722} C_DIS
LIN {X 2.3748,Y 4.1155,Z 37,A -2.4316,B 0,C 0,E1 0.1598,E2 90.0722} C_DIS
LIN {X 2.9236,Y 3.7438,Z 37,A -2.4272,B 0,C 0,E1 0.1598,E2 90.0722} C_DIS
LIN {X 3.4167,Y 3.3009,Z 37,A -2.4278,B 0,C 0,E1 0.1598,E2 90.0722} C_DIS
LIN {X 3.8425,Y 2.7929,Z 37,A -2.4337,B 0,C 0,E1 0.1598,E2 90.0722} C_DIS
LIN {X 4.1939,Y 2.231,Z 37,A -2.4446,B 0,C 0,E1 0.1598,E2 90.0722} C_DIS
LIN {X 4.4648,Y 1.626,Z 37,A -2.4603,B 0,C 0,E1 0.1598,E2 90.0721} C_DIS
LIN {X 4.6459,Y 0.9884,Z 37,A -2.4807,B 0,C 0,E1 0.1598,E2 90.0721} C_DIS
LIN {X 4.7399,Y 0.3324,Z 37,A -2.5052,B 0,C 0,E1 0.1598,E2 90.072} C_DIS
LIN {X 4.7393,Y -0.3305,Z 37,A -2.5334,B 0,C 0,E1 0.1598,E2 90.072} C_DIS
LIN {X 4.6483,Y -0.987,Z 37,A -2.5647,B 0,C 0,E1 0.1598,E2 90.072} C_DIS
LIN {X 4.4654,Y -1.6242,Z 37,A -2.5986,B 0,C 0,E1 0.1598,E2 90.0719} C_DIS
LIN {X 4.1967,Y -2.2303,Z 37,A -2.6343,B 0,C 0,E1 0.1598,E2 90.0719} C_DIS
LIN {X 3.8431,Y -2.791,Z 37,A -2.6712,B 0,C 0,E1 0.1598,E2 90.0719} C_DIS
LIN {X 3.4172,Y -3.2987,Z 37,A -2.7085,B 0,C 0,E1 0.1598,E2 90.0719} C_DIS
LIN {X 2.9264,Y -3.7444,Z 37,A -2.7455,B 0,C 0,E1 0.1598,E2 90.0719} C_DIS
LIN {X 2.3769,Y -4.1154,Z 37,A -2.7815,B 0,C 0,E1 0.1598,E2 90.0718} C_DIS
LIN {X 1.7809,Y -4.4059,Z 37,A -2.8158,B 0,C 0,E1 0.1598,E2 90.0718} C_DIS
LIN {X 1.1506,Y -4.6115,Z 37,A -2.8477,B 0,C 0,E1 0.1598,E2 90.0718} C_DIS
LIN {X 0.4977,Y -4.7269,Z 37,A -2.8766,B 0,C 0,E1 0.1598,E2 90.0718} C_DIS
LIN {X 0.4977,Y -4.7269,Z 37,A -2.8766,B 0,C 0,E1 0.1598,E2 90.0718} C_DIS
Enddeposition()
LIN {X 0.0309,Y -5.687,Z 37,A -2.9334,B 0,C 0,E1 0.1598,E2 90.0705} C_DIS
Startdeposition()
$VEL.CP = VEL_PRINT
LIN {X 0.6546,Y -5.647,Z 37,A -2.91,B 0,C 0,E1 0.1598,E2 90.0716} C_DIS
LIN {X 1.4722,Y -5.4894,Z 37,A -2.8733,B 0,C 0,E1 0.1598,E2 90.0717} C_DIS
LIN {X 2.2585,Y -5.2158,Z 37,A -2.8328,B 0,C 0,E1 0.1598,E2 90.0717} C_DIS
LIN {X 2.9956,Y -4.8288,Z 37,A -2.7892,B 0,C 0,E1 0.1598,E2 90.0717} C_DIS
LIN {X 3.6691,Y -4.3394,Z 37,A -2.7436,B 0,C 0,E1 0.1598,E2 90.0717} C_DIS
LIN {X 4.2633,Y -3.7564,Z 37,A -2.6969,B 0,C 0,E1 0.1598,E2 90.0718} C_DIS
LIN {X 4.7668,Y -3.0935,Z 37,A -2.6501,B 0,C 0,E1 0.1598,E2 90.0718} C_DIS
LIN {X 5.1675,Y -2.3638,Z 37,A -2.6043,B 0,C 0,E1 0.1598,E2 90.0718} C_DIS
LIN {X 5.4598,Y -1.584,Z 37,A -2.5603,B 0,C 0,E1 0.1598,E2 90.0718} C_DIS
LIN {X 5.6318,Y -0.7693,Z 37,A -2.5192,B 0,C 0,E1 0.1598,E2 90.0718} C_DIS
LIN {X 5.6857,Y 0.0618,Z 37,A -2.4818,B 0,C 0,E1 0.1598,E2 90.0718} C_DIS
LIN {X 5.6146,Y 0.8916,Z 37,A -2.4491,B 0,C 0,E1 0.1598,E2 90.0719} C_DIS
LIN {X 5.4239,Y 1.7022,Z 37,A -2.4216,B 0,C 0,E1 0.1598,E2 90.0719} C_DIS
LIN {X 5.1166,Y 2.4762,Z 37,A -2.4,B 0,C 0,E1 0.1598,E2 90.072} C_DIS
LIN {X 4.7013,Y 3.1981,Z 37,A -2.3846,B 0,C 0,E1 0.1598,E2 90.072} C_DIS
LIN {X 4.183,Y 3.8501,Z 37,A -2.376,B 0,C 0,E1 0.1598,E2 90.0721} C_DIS
LIN {X 3.5752,Y 4.4195,Z 37,A -2.3743,B 0,C 0,E1 0.1598,E2 90.0722} C_DIS
LIN {X 2.8906,Y 4.8935,Z 37,A -2.3794,B 0,C 0,E1 0.1598,E2 90.0722} C_DIS
LIN {X 2.1455,Y 5.2655,Z 37,A -2.3912,B 0,C 0,E1 0.1598,E2 90.0722} C_DIS
LIN {X 1.0639,Y 5.5902,Z 37,A -2.4173,B 0,C 0,E1 0.1598,E2 90.0722} C_DIS
LIN {X 0.1813,Y 5.6814,Z 37,A -2.446,B 0,C 0,E1 0.1598,E2 90.0722} C_DIS
LIN {X -0.5281,Y 5.6607,Z 37,A -2.4731,B 0,C 0,E1 0.1598,E2 90.0722} C_DIS
LIN {X -1.2291,Y 5.5499,Z 37,A -2.5036,B 0,C 0,E1 0.1598,E2 90.0722} C_DIS
LIN {X -2.0795,Y 5.2972,Z 37,A -2.5457,B 0,C 0,E1 0.1598,E2 90.0722} C_DIS
LIN {X -3.4598,Y 4.5163,Z 37,A -2.6293,B 0,C 0,E1 0.1598,E2 90.0717} C_DIS
LIN {X -4.1508,Y 3.8822,Z 37,A -2.6817,B 0,C 0,E1 0.1598,E2 90.0718} C_DIS
LIN {X -4.626,Y 3.3019,Z 37,A -2.7238,B 0,C 0,E1 0.1598,E2 90.0718} C_DIS
LIN {X -5.0221,Y 2.6646,Z 37,A -2.7653,B 0,C 0,E1 0.1598,E2 90.0717} C_DIS
LIN {X -5.4358,Y 1.6799,Z 37,A -2.8219,B 0,C 0,E1 0.1598,E2 90.0713} C_DIS
LIN {X -5.6875,Y 0.1619,Z 37,A -2.8947,B 0,C 0,E1 0.1598,E2 90.0705} C_DIS
LIN {X -5.6152,Y -0.8835,Z 37,A -2.9369,B 0,C 0,E1 0.1598,E2 90.0711} C_DIS
LIN {X -5.4241,Y -1.6998,Z 37,A -2.9646,B 0,C 0,E1 0.1598,E2 90.0713} C_DIS
LIN {X -5.1165,Y -2.4799,Z 37,A -2.9864,B 0,C 0,E1 0.1598,E2 90.0713} C_DIS
LIN {X -4.6952,Y -3.2049,Z 37,A -3.0017,B 0,C 0,E1 0.1598,E2 90.0713} C_DIS
LIN {X -4.1727,Y -3.8606,Z 37,A -3.0103,B 0,C 0,E1 0.1598,E2 90.0713} C_DIS
LIN {X -3.7235,Y -4.3015,Z 37,A -3.0127,B 0,C 0,E1 0.1598,E2 90.0715} C_DIS
LIN {X -3.0876,Y -4.7736,Z 37,A -3.0093,B 0,C 0,E1 0.1598,E2 90.0715} C_DIS
LIN {X -2.5056,Y -5.1079,Z 37,A -3.0022,B 0,C 0,E1 0.1598,E2 90.0715} C_DIS
LIN {X -1.3133,Y -5.5372,Z 37,A -2.9767,B 0,C 0,E1 0.1598,E2 90.0715} C_DIS
LIN {X -0.4765,Y -5.6642,Z 37,A -2.9514,B 0,C 0,E1 0.1598,E2 90.0716} C_DIS
LIN {X -0.4765,Y -5.6642,Z 37,A -2.9514,B 0,C 0,E1 0.1598,E2 90.0716} C_DIS
Enddeposition()
LIN {X 0.0389,Y -6.6206,Z 37,A -2.9722,B 0,C 0,E1 0.1598,E2 90.0704} C_DIS
Startdeposition()
$VEL.CP = VEL_PRINT
LIN {X -0.8348,Y -6.5669,Z 37,A -3.003,B 0,C 0,E1 0.1598,E2 90.0715} C_DIS
LIN {X -1.524,Y -6.4418,Z 37,A -3.0231,B 0,C 0,E1 0.1598,E2 90.0715} C_DIS
LIN {X -2.1965,Y -6.2461,Z 37,A -3.0394,B 0,C 0,E1 0.1598,E2 90.0715} C_DIS
LIN {X -3.1378,Y -5.8327,Z 37,A -3.0563,B 0,C 0,E1 0.1598,E2 90.0714} C_DIS
LIN {X -3.8668,Y -5.3722,Z 37,A -3.0635,B 0,C 0,E1 0.1598,E2 90.0714} C_DIS
LIN {X -4.4047,Y -4.9404,Z 37,A -3.0649,B 0,C 0,E1 0.1598,E2 90.0714} C_DIS
LIN {X -4.8956,Y -4.4561,Z 37,A -3.0624,B 0,C 0,E1 0.1598,E2 90.0714} C_DIS
LIN {X -5.3321,Y -3.9219,Z 37,A -3.0558,B 0,C 0,E1 0.1598,E2 90.0714} C_DIS
LIN {X -5.7114,Y -3.3458,Z 37,A -3.0453,B 0,C 0,E1 0.1598,E2 90.0714} C_DIS
LIN {X -6.0295,Y -2.7339,Z 37,A -3.031,B 0,C 0,E1 0.1598,E2 90.0714} C_DIS
LIN {X -6.2817,Y -2.092,Z 37,A -3.0131,B 0,C 0,E1 0.1598,E2 90.0714} C_DIS
LIN {X -6.4658,Y -1.4273,Z 37,A -2.9917,B 0,C 0,E1 0.1598,E2 90.0714} C_DIS
LIN {X -6.5763,Y -0.7465,Z 37,A -2.9669,B 0,C 0,E1 0.1598,E2 90.0714} C_DIS
LIN {X -6.6188,Y -0.058,Z 37,A -2.9394,B 0,C 0,E1 0.1598,E2 90.0714} C_DIS
LIN {X -6.59,Y 0.6311,Z 37,A -2.9092,B 0,C 0,E1 0.1598,E2 90.0714} C_DIS
LIN {X -6.4902,Y 1.3136,Z 37,A -2.8766,B 0,C 0,E1 0.1598,E2 90.0714} C_DIS
LIN {X -6.319,Y 1.9819,Z 37,A -2.8421,B 0,C 0,E1 0.1598,E2 90.0716} C_DIS
LIN {X -6.0752,Y 2.6272,Z 37,A -2.8058,B 0,C 0,E1 0.1598,E2 90.0716} C_DIS
LIN {X -5.7688,Y 3.2451,Z 37,A -2.7684,B 0,C 0,E1 0.1598,E2 90.0716} C_DIS
LIN {X -5.3998,Y 3.8278,Z 37,A -2.7302,B 0,C 0,E1 0.1598,E2 90.0718} C_DIS
LIN {X -4.9717,Y 4.3686,Z 37,A -2.6916,B 0,C 0,E1 0.1598,E2 90.0718} C_DIS
LIN {X -4.4903,Y 4.8625,Z 37,A -2.653,B 0,C 0,E1 0.1598,E2 90.0719} C_DIS
LIN {X -3.96,Y 5.3034,Z 37,A -2.6148,B 0,C 0,E1 0.1598,E2 90.0719} C_DIS
LIN {X -3.3866,Y 5.6869,Z 37,A -2.5775,B 0,C 0,E1 0.1598,E2 90.0721} C_DIS
LIN {X -2.7767,Y 6.0088,Z 37,A -2.5414,B 0,C 0,E1 0.1598,E2 90.0721} C_DIS
LIN {X -2.1365,Y 6.2656,Z 37,A -2.5069,B 0,C 0,E1 0.1598,E2 90.0721} C_DIS
LIN {X -1.3049,Y 6.4936,Z 37,A -2.4666,B 0,C 0,E1 0.1598,E2 90.0723} C_DIS
LIN {X -0.1519,Y 6.6173,Z 37,A -2.4188,B 0,C 0,E1 0.1598,E2 90.0723} C_DIS
LIN {X 1.0075,Y 6.5463,Z 37,A -2.379,B 0,C 0,E1 0.1598,E2 90.0723} C_DIS
LIN {X 1.9015,Y 6.3413,Z 37,A -2.3547,B 0,C 0,E1 0.1598,E2 90.0724} C_DIS
LIN {X 2.5916,Y 6.092,Z 37,A -2.3399,B 0,C 0,E1 0.1598,E2 90.0724} C_DIS
LIN {X 3.2486,Y 5.7659,Z 37,A -2.3294,B 0,C 0,E1 0.1598,E2 90.0724} C_DIS
LIN {X 3.8679,Y 5.3724,Z 37,A -2.3233,B 0,C 0,E1 0.1598,E2 90.0724} C_DIS
LIN {X 4.4388,Y 4.9114,Z 37,A -2.3218,B 0,C 0,E1 0.1598,E2 90.0724} C_DIS
LIN {X 4.9552,Y 4.3901,Z 37,A -2.3249,B 0,C 0,E1 0.1598,E2 90.0724} C_DIS
LIN {X 5.4106,Y 3.8147,Z 37,A -2.3325,B 0,C 0,E1 0.1598,E2 90.0723} C_DIS
LIN {X 5.8011,Y 3.1936,Z 37,A -2.3446,B 0,C 0,E1 0.1598,E2 90.0723} C_DIS
LIN {X 6.1176,Y 2.5317,Z 37,A -2.361,B 0,C 0,E1 0.1598,E2 90.0722} C_DIS
LIN {X 6.3595,Y 1.8389,Z 37,A -2.3816,B 0,C 0,E1 0.1598,E2 90.0722} C_DIS
LIN {X 6.5748,Y 0.8011,Z 37,A -2.4176,B 0,C 0,E1 0.1598,E2 90.0718} C_DIS
LIN {X 6.6164,Y -0.1178,Z 37,A -2.4553,B 0,C 0,E1 0.1598,E2 90.0718} C_DIS
LIN {X 6.5631,Y -0.8515,Z 37,A -2.4887,B 0,C 0,E1 0.1598,E2 90.0719} C_DIS
LIN {X 6.4285,Y -1.5748,Z 37,A -2.5245,B 0,C 0,E1 0.1598,E2 90.0719} C_DIS
LIN {X 6.2154,Y -2.2791,Z 37,A -2.5624,B 0,C 0,E1 0.1598,E2 90.0719} C_DIS
LIN {X 5.9226,Y -2.9543,Z 37,A -2.6019,B 0,C 0,E1 0.1598,E2 90.0719} C_DIS
LIN {X 5.5583,Y -3.5936,Z 37,A -2.6426,B 0,C 0,E1 0.1598,E2 90.0719} C_DIS
LIN {X 5.1251,Y -4.1884,Z 37,A -2.6839,B 0,C 0,E1 0.1598,E2 90.0719} C_DIS
LIN {X 4.6278,Y -4.7304,Z 37,A -2.7252,B 0,C 0,E1 0.1598,E2 90.0718} C_DIS
LIN {X 4.0743,Y -5.2152,Z 37,A -2.7662,B 0,C 0,E1 0.1598,E2 90.0718} C_DIS
LIN {X 3.4705,Y -5.6358,Z 37,A -2.8063,B 0,C 0,E1 0.1598,E2 90.0718} C_DIS
LIN {X 2.8235,Y -5.9862,Z 37,A -2.845,B 0,C 0,E1 0.1598,E2 90.0718} C_DIS
LIN {X 2.1417,Y -6.2631,Z 37,A -2.8818,B 0,C 0,E1 0.1598,E2 90.0717} C_DIS
LIN {X 1.1067,Y -6.5303,Z 37,A -2.9312,B 0,C 0,E1 0.1598,E2 90.0717} C_DIS
LIN {X 0.0389,Y -6.6206,Z 37,A -2.9742,B 0,C 0,E1 0.1598,E2 90.0717} C_DIS
Enddeposition()
LIN {X 0.0389,Y -6.6206,Z 37,A -2.9742,B 0,C 0,E1 0.1598,E2 90.0717} C_DIS
Startdeposition()
$VEL.CP = VEL_PRINT
LIN {X 0.7352,Y -7.5177,Z 37,A -2.9864,B 0,C 0,E1 0.1598,E2 90.071} C_DIS
LIN {X 1.4891,Y -7.4088,Z 37,A -2.9547,B 0,C 0,E1 0.1598,E2 90.0716} C_DIS
LIN {X 2.6992,Y -7.0588,Z 37,A -2.8954,B 0,C 0,E1 0.1598,E2 90.0716} C_DIS
LIN {X 3.7624,Y -6.5482,Z 37,A -2.8346,B 0,C 0,E1 0.1598,E2 90.0716} C_DIS
LIN {X 4.6677,Y -5.9428,Z 37,A -2.7755,B 0,C 0,E1 0.1598,E2 90.0716} C_DIS
LIN {X 5.3392,Y -5.3502,Z 37,A -2.7257,B 0,C 0,E1 0.1598,E2 90.0718} C_DIS
LIN {X 6.1885,Y -4.3363,Z 37,A -2.6508,B 0,C 0,E1 0.1598,E2 90.0714} C_DIS
LIN {X 6.8762,Y -3.1375,Z 37,A -2.5743,B 0,C 0,E1 0.1598,E2 90.0714} C_DIS
LIN {X 7.2318,Y -2.1927,Z 37,A -2.5211,B 0,C 0,E1 0.1598,E2 90.0717} C_DIS
LIN {X 7.4945,Y -0.9434,Z 37,A -2.4578,B 0,C 0,E1 0.1598,E2 90.0714} C_DIS
LIN {X 7.5544,Y -0.1995,Z 37,A -2.4243,B 0,C 0,E1 0.1598,E2 90.0719} C_DIS
LIN {X 7.5275,Y 0.6848,Z 37,A -2.3876,B 0,C 0,E1 0.1598,E2 90.0719} C_DIS
LIN {X 7.3784,Y 1.6341,Z 37,A -2.3526,B 0,C 0,E1 0.1598,E2 90.0719} C_DIS
LIN {X 7.1671,Y 2.3995,Z 37,A -2.3279,B 0,C 0,E1 0.1598,E2 90.0721} C_DIS
LIN {X 6.2093,Y 4.3063,Z 37,A -2.2813,B 0,C 0,E1 0.1598,E2 90.0715} C_DIS
LIN {X 5.3208,Y 5.3679,Z 37,A -2.2693,B 0,C 0,E1 0.1598,E2 90.0719} C_DIS
LIN {X 4.4553,Y 6.0989,Z 37,A -2.2704,B 0,C 0,E1 0.1598,E2 90.0722} C_DIS
LIN {X 3.7672,Y 6.5462,Z 37,A -2.277,B 0,C 0,E1 0.1598,E2 90.0724} C_DIS
LIN {X 2.748,Y 7.0408,Z 37,A -2.2936,B 0,C 0,E1 0.1598,E2 90.0724} C_DIS
LIN {X 1.4565,Y 7.4157,Z 37,A -2.3254,B 0,C 0,E1 0.1598,E2 90.0724} C_DIS
LIN {X 0.4394,Y 7.5444,Z 37,A -2.3576,B 0,C 0,E1 0.1598,E2 90.0724} C_DIS
LIN {X -0.7986,Y 7.5113,Z 37,A -2.4047,B 0,C 0,E1 0.1598,E2 90.0724} C_DIS
LIN {X -1.7632,Y 7.3495,Z 37,A -2.4471,B 0,C 0,E1 0.1598,E2 90.0723} C_DIS
LIN {X -2.9358,Y 6.963,Z 37,A -2.5067,B 0,C 0,E1 0.1598,E2 90.0722} C_DIS
LIN {X -3.6909,Y 6.594,Z 37,A -2.5501,B 0,C 0,E1 0.1598,E2 90.0721} C_DIS
LIN {X -4.6915,Y 5.9245,Z 37,A -2.6152,B 0,C 0,E1 0.1598,E2 90.0719} C_DIS
LIN {X -5.4387,Y 5.2463,Z 37,A -2.6714,B 0,C 0,E1 0.1598,E2 90.0717} C_DIS
LIN {X -6.1131,Y 4.4454,Z 37,A -2.73,B 0,C 0,E1 0.1598,E2 90.0717} C_DIS
LIN {X -6.5413,Y 3.7868,Z 37,A -2.7738,B 0,C 0,E1 0.1598,E2 90.0717} C_DIS
LIN {X -7.1292,Y 2.5076,Z 37,A -2.8489,B 0,C 0,E1 0.1598,E2 90.071} C_DIS
LIN {X -7.3667,Y 1.6898,Z 37,A -2.8925,B 0,C 0,E1 0.1598,E2 90.0712} C_DIS
LIN {X -7.5357,Y 0.5282,Z 37,A -2.9476,B 0,C 0,E1 0.1598,E2 90.0709} C_DIS
LIN {X -7.5516,Y -0.3239,Z 37,A -2.9843,B 0,C 0,E1 0.1598,E2 90.0709} C_DIS
LIN {X -7.4487,Y -1.2757,Z 37,A -3.0208,B 0,C 0,E1 0.1598,E2 90.071} C_DIS
LIN {X -7.2141,Y -2.2494,Z 37,A -3.0534,B 0,C 0,E1 0.1598,E2 90.071} C_DIS
LIN {X -6.7631,Y -3.3611,Z 37,A -3.0837,B 0,C 0,E1 0.1598,E2 90.0708} C_DIS
LIN {X -6.3477,Y -4.0927,Z 37,A -3.0998,B 0,C 0,E1 0.1598,E2 90.0711} C_DIS
LIN {X -5.8536,Y -4.7736,Z 37,A -3.1105,B 0,C 0,E1 0.1598,E2 90.0711} C_DIS
LIN {X -5.2854,Y -5.394,Z 37,A -3.116,B 0,C 0,E1 0.1598,E2 90.0712} C_DIS
LIN {X -4.6523,Y -5.9478,Z 37,A -3.1163,B 0,C 0,E1 0.1598,E2 90.0712} C_DIS
LIN {X -3.7849,Y -6.5423,Z 37,A -3.1097,B 0,C 0,E1 0.1598,E2 90.0712} C_DIS
LIN {X -2.7812,Y -7.0223,Z 37,A -3.0933,B 0,C 0,E1 0.1598,E2 90.0713} C_DIS
LIN {X -1.8546,Y -7.3257,Z 37,A -3.0723,B 0,C 0,E1 0.1598,E2 90.0714} C_DIS
LIN {X -0.7978,Y -7.5148,Z 37,A -3.0416,B 0,C 0,E1 0.1598,E2 90.0714} C_DIS
LIN {X 0.0717,Y -7.5559,Z 37,A -3.0115,B 0,C 0,E1 0.1598,E2 90.0716} C_DIS
Enddeposition()
LIN {X 0.0717,Y -7.5559,Z 37,A -3.0115,B 0,C 0,E1 0.1598,E2 90.0716} C_DIS
Startdeposition()
$VEL.CP = VEL_PRINT
LIN {X -0.5399,Y -8.4682,Z 37,A -3.0724,B 0,C 0,E1 0.1598,E2 90.0709} C_DIS
LIN {X -1.3723,Y -8.3735,Z 37,A -3.0994,B 0,C 0,E1 0.1598,E2 90.0714} C_DIS
LIN {X -2.1914,Y -8.1975,Z 37,A -3.1219,B 0,C 0,E1 0.1598,E2 90.0714} C_DIS
LIN {X -2.9893,Y -7.9423,Z 37,A -3.1403,B 0,C 0,E1 0.1598,E2 90.0714} C_DIS
LIN {X -3.7576,Y -7.6085,Z 37,A -3.1543,B 0,C 0,E1 0.1598,E2 90.0714} C_DIS
LIN {X -4.4895,Y -7.2008,Z 37,A -3.1638,B 0,C 0,E1 0.1598,E2 90.0713} C_DIS
LIN {X -5.1776,Y -6.7229,Z 37,A -3.1687,B 0,C 0,E1 0.1598,E2 90.0713} C_DIS
LIN {X -5.8153,Y -6.1795,Z 37,A -3.169,B 0,C 0,E1 0.1598,E2 90.0712} C_DIS
LIN {X -6.3963,Y -5.576,Z 37,A -3.1647,B 0,C 0,E1 0.1598,E2 90.0712} C_DIS
LIN {X -6.9152,Y -4.9182,Z 37,A -3.1559,B 0,C 0,E1 0.1598,E2 90.0712} C_DIS
LIN {X -7.3668,Y -4.2125,Z 37,A -3.1425,B 0,C 0,E1 0.1598,E2 90.0712} C_DIS
LIN {X -7.7467,Y -3.4656,Z 37,A -3.1249,B 0,C 0,E1 0.1598,E2 90.0712} C_DIS
LIN {X -8.051,Y -2.685,Z 37,A -3.103,B 0,C 0,E1 0.1598,E2 90.0712} C_DIS
LIN {X -8.277,Y -1.8781,Z 37,A -3.0771,B 0,C 0,E1 0.1598,E2 90.0712} C_DIS
LIN {X -8.4226,Y -1.0528,Z 37,A -3.0476,B 0,C 0,E1 0.1598,E2 90.0712} C_DIS
LIN {X -8.4896,Y 0.1375,Z 37,A -2.9994,B 0,C 0,E1 0.1598,E2 90.0709} C_DIS
LIN {X -8.4051,Y 1.1718,Z 37,A -2.9528,B 0,C 0,E1 0.1598,E2 90.0711} C_DIS
LIN {X -8.2509,Y 1.9877,Z 37,A -2.9128,B 0,C 0,E1 0.1598,E2 90.0713} C_DIS
LIN {X -8.0174,Y 2.7845,Z 37,A -2.8706,B 0,C 0,E1 0.1598,E2 90.0714} C_DIS
LIN {X -7.7067,Y 3.5545,Z 37,A -2.8266,B 0,C 0,E1 0.1598,E2 90.0714} C_DIS
LIN {X -7.3221,Y 4.2903,Z 37,A -2.7814,B 0,C 0,E1 0.1598,E2 90.0716} C_DIS
LIN {X -6.8675,Y 4.9849,Z 37,A -2.7353,B 0,C 0,E1 0.1598,E2 90.0716} C_DIS
LIN {X -6.3471,Y 5.6319,Z 37,A -2.6888,B 0,C 0,E1 0.1598,E2 90.0718} C_DIS
LIN {X -5.7662,Y 6.2249,Z 37,A -2.6424,B 0,C 0,E1 0.1598,E2 90.0718} C_DIS
LIN {X -5.1302,Y 6.7584,Z 37,A -2.5964,B 0,C 0,E1 0.1598,E2 90.072} C_DIS
LIN {X -4.4451,Y 7.2273,Z 37,A -2.5514,B 0,C 0,E1 0.1598,E2 90.072} C_DIS
LIN {X -3.7176,Y 7.6272,Z 37,A -2.5076,B 0,C 0,E1 0.1598,E2 90.0722} C_DIS
LIN {X -2.5408,Y 8.1011,Z 37,A -2.4441,B 0,C 0,E1 0.1598,E2 90.0722} C_DIS
LIN {X -1.5015,Y 8.3539,Z 37,A -2.3951,B 0,C 0,E1 0.1598,E2 90.0723} C_DIS
LIN {X -0.4394,Y 8.4802,Z 37,A -2.3506,B 0,C 0,E1 0.1598,E2 90.0724} C_DIS
LIN {X 0.7465,Y 8.4549,Z 37,A -2.3078,B 0,C 0,E1 0.1598,E2 90.0724} C_DIS
LIN {X 1.59,Y 8.3375,Z 37,A -2.2817,B 0,C 0,E1 0.1598,E2 90.0725} C_DIS
LIN {X 2.4176,Y 8.1364,Z 37,A -2.2596,B 0,C 0,E1 0.1598,E2 90.0725} C_DIS
LIN {X 3.2207,Y 7.8533,Z 37,A -2.242,B 0,C 0,E1 0.1598,E2 90.0725} C_DIS
LIN {X 3.9914,Y 7.491,Z 37,A -2.2289,B 0,C 0,E1 0.1598,E2 90.0725} C_DIS
LIN {X 4.9857,Y 6.8745,Z 37,A -2.2182,B 0,C 0,E1 0.1598,E2 90.0724} C_DIS
LIN {X 5.9626,Y 6.0395,Z 37,A -2.2175,B 0,C 0,E1 0.1598,E2 90.0722} C_DIS
LIN {X 6.5504,Y 5.3958,Z 37,A -2.2233,B 0,C 0,E1 0.1598,E2 90.0723} C_DIS
LIN {X 7.0694,Y 4.6955,Z 37,A -2.234,B 0,C 0,E1 0.1598,E2 90.0723} C_DIS
LIN {X 7.514,Y 3.9457,Z 37,A -2.2495,B 0,C 0,E1 0.1598,E2 90.0723} C_DIS
LIN {X 7.8794,Y 3.1543,Z 37,A -2.2697,B 0,C 0,E1 0.1598,E2 90.0722} C_DIS
LIN {X 8.1614,Y 2.3294,Z 37,A -2.2944,B 0,C 0,E1 0.1598,E2 90.0722} C_DIS
LIN {X 8.4077,Y 1.1928,Z 37,A -2.3335,B 0,C 0,E1 0.1598,E2 90.0718} C_DIS
LIN {X 8.4922,Y -0.0068,Z 37,A -2.3815,B 0,C 0,E1 0.1598,E2 90.0716} C_DIS
LIN {X 8.4204,Y -1.0972,Z 37,A -2.4308,B 0,C 0,E1 0.1598,E2 90.0716} C_DIS
LIN {X 8.174,Y -2.2839,Z 37,A -2.4903,B 0,C 0,E1 0.1598,E2 90.0714} C_DIS
LIN {X 7.8964,Y -3.1096,Z 37,A -2.5361,B 0,C 0,E1 0.1598,E2 90.0718} C_DIS
LIN {X 7.5357,Y -3.9024,Z 37,A -2.5833,B 0,C 0,E1 0.1598,E2 90.0718} C_DIS
LIN {X 7.0958,Y -4.6541,Z 37,A -2.6315,B 0,C 0,E1 0.1598,E2 90.0718} C_DIS
LIN {X 6.5815,Y -5.357,Z 37,A -2.6804,B 0,C 0,E1 0.1598,E2 90.0718} C_DIS
LIN {X 5.9978,Y -6.0035,Z 37,A -2.7295,B 0,C 0,E1 0.1598,E2 90.0718} C_DIS
LIN {X 5.351,Y -6.5869,Z 37,A -2.7781,B 0,C 0,E1 0.1598,E2 90.0717} C_DIS
LIN {X 4.6479,Y -7.101,Z 37,A -2.8258,B 0,C 0,E1 0.1598,E2 90.0717} C_DIS
LIN {X 3.584,Y -7.6978,Z 37,A -2.8903,B 0,C 0,E1 0.1598,E2 90.0716} C_DIS
LIN {X 2.5235,Y -8.1066,Z 37,A -2.9466,B 0,C 0,E1 0.1598,E2 90.0716} C_DIS
LIN {X 1.5225,Y -8.3496,Z 37,A -2.9937,B 0,C 0,E1 0.1598,E2 90.0716} C_DIS
LIN {X 0.7057,Y -8.4581,Z 37,A -3.0283,B 0,C 0,E1 0.1598,E2 90.0716} C_DIS
LIN {X 0.7057,Y -8.4581,Z 37,A -3.0283,B 0,C 0,E1 0.1598,E2 90.0716} C_DIS
Enddeposition()
LIN {X 0.0009,Y -4.7563,Z 38,A -2.882,B 0,C 0,E1 0.1598,E2 90.0604} C_DIS
Startdeposition()
$VEL.CP = VEL_PRINT
LIN {X 0.0009,Y -4.7563,Z 38,A -2.8877,B 0,C 0,E1 0.1598,E2 90.0661} C_DIS
LIN {X 0.8261,Y -4.6807,Z 38,A -2.8591,B 0,C 0,E1 0.1598,E2 90.0711} C_DIS
LIN {X 1.4694,Y -4.52,Z 38,A -2.8292,B 0,C 0,E1 0.1598,E2 90.0718} C_DIS
LIN {X 2.0841,Y -4.2714,Z 38,A -2.7961,B 0,C 0,E1 0.1598,E2 90.0718} C_DIS
LIN {X 2.6583,Y -3.9396,Z 38,A -2.7609,B 0,C 0,E1 0.1598,E2 90.0718} C_DIS
LIN {X 3.1796,Y -3.53,Z 38,A -2.7243,B 0,C 0,E1 0.1598,E2 90.0718} C_DIS
LIN {X 3.7425,Y -2.9228,Z 38,A -2.6776,B 0,C 0,E1 0.1598,E2 90.0718} C_DIS
LIN {X 4.0305,Y -2.5173,Z 38,A -2.6499,B 0,C 0,E1 0.1598,E2 90.0719} C_DIS
LIN {X 4.3408,Y -1.9316,Z 38,A -2.6135,B 0,C 0,E1 0.1598,E2 90.0719} C_DIS
LIN {X 4.5679,Y -1.3088,Z 38,A -2.5786,B 0,C 0,E1 0.1598,E2 90.0719} C_DIS
LIN {X 4.7062,Y -0.6605,Z 38,A -2.5458,B 0,C 0,E1 0.1598,E2 90.0719} C_DIS
LIN {X 4.7508,Y 0.001,Z 38,A -2.516,B 0,C 0,E1 0.1598,E2 90.0719} C_DIS
LIN {X 4.7045,Y 0.662,Z 38,A -2.4896,B 0,C 0,E1 0.1598,E2 90.072} C_DIS
LIN {X 4.5665,Y 1.3104,Z 38,A -2.4671,B 0,C 0,E1 0.1598,E2 90.072} C_DIS
LIN {X 4.339,Y 1.9328,Z 38,A -2.449,B 0,C 0,E1 0.1598,E2 90.072} C_DIS
LIN {X 4.029,Y 2.5187,Z 38,A -2.4355,B 0,C 0,E1 0.1598,E2 90.0721} C_DIS
LIN {X 3.6381,Y 3.054,Z 38,A -2.4271,B 0,C 0,E1 0.1598,E2 90.0721} C_DIS
LIN {X 3.1778,Y 3.5308,Z 38,A -2.4239,B 0,C 0,E1 0.1598,E2 90.0722} C_DIS
LIN {X 2.6555,Y 3.9389,Z 38,A -2.4258,B 0,C 0,E1 0.1598,E2 90.0722} C_DIS
LIN {X 2.0822,Y 4.2715,Z 38,A -2.4328,B 0,C 0,E1 0.1598,E2 90.0722} C_DIS
LIN {X 1.4672,Y 4.5191,Z 38,A -2.445,B 0,C 0,E1 0.1598,E2 90.0722} C_DIS
LIN {X 0.824,Y 4.6794,Z 38,A -2.462,B 0,C 0,E1 0.1598,E2 90.0722} C_DIS
LIN {X 0.1649,Y 4.749,Z 38,A -2.4833,B 0,C 0,E1 0.1598,E2 90.0722} C_DIS
LIN {X -0.4976,Y 4.7254,Z 38,A -2.5087,B 0,C 0,E1 0.1598,E2 90.0722} C_DIS
LIN {X -1.1509,Y 4.6118,Z 38,A -2.5376,B 0,C 0,E1 0.1598,E2 90.0722} C_DIS
LIN {X -1.7812,Y 4.4061,Z 38,A -2.5696,B 0,C 0,E1 0.1598,E2 90.0722} C_DIS
LIN {X -2.3769,Y 4.1152,Z 38,A -2.6038,B 0,C 0,E1 0.1598,E2 90.0721} C_DIS
LIN {X -2.9266,Y 3.7445,Z 38,A -2.6397,B 0,C 0,E1 0.1598,E2 90.072} C_DIS
LIN {X -3.4186,Y 3.3001,Z 38,A -2.6767,B 0,C 0,E1 0.1598,E2 90.072} C_DIS
LIN {X -3.8447,Y 2.7922,Z 38,A -2.7138,B 0,C 0,E1 0.1598,E2 90.0718} C_DIS
LIN {X -4.1968,Y 2.2305,Z 38,A -2.7505,B 0,C 0,E1 0.1598,E2 90.0718} C_DIS
LIN {X -4.4652,Y 1.6242,Z 38,A -2.7861,B 0,C 0,E1 0.1598,E2 90.0717} C_DIS
LIN {X -4.6478,Y 0.987,Z 38,A -2.8197,B 0,C 0,E1 0.1598,E2 90.0717} C_DIS
LIN {X -4.7388,Y 0.3306,Z 38,A -2.8509,B 0,C 0,E1 0.1598,E2 90.0715} C_DIS
LIN {X -4.74,Y -0.3323,Z 38,A -2.879,B 0,C 0,E1 0.1598,E2 90.0715} C_DIS
LIN {X -4.6468,Y -0.9885,Z 38,A -2.9033,B 0,C 0,E1 0.1598,E2 90.0715} C_DIS
LIN {X -4.4631,Y -1.6252,Z 38,A -2.9236,B 0,C 0,E1 0.1598,E2 90.0715} C_DIS
LIN {X -4.1957,Y -2.2319,Z 38,A -2.9395,B 0,C 0,E1 0.1598,E2 90.0715} C_DIS
LIN {X -3.8417,Y -2.7922,Z 38,A -2.9502,B 0,C 0,E1 0.1598,E2 90.0715} C_DIS
LIN {X -3.4167,Y -3.3008,Z 38,A -2.9562,B 0,C 0,E1 0.1598,E2 90.0715} C_DIS
LIN {X -2.9237,Y -3.7438,Z 38,A -2.9569,B 0,C 0,E1 0.1598,E2 90.0715} C_DIS
LIN {X -2.3744,Y -4.1147,Z 38,A -2.9525,B 0,C 0,E1 0.1598,E2 90.0715} C_DIS
LIN {X -1.7789,Y -4.4055,Z 38,A -2.9431,B 0,C 0,E1 0.1598,E2 90.0716} C_DIS
LIN {X -1.1484,Y -4.6098,Z 38,A -2.9286,B 0,C 0,E1 0.1598,E2 90.0716} C_DIS
LIN {X -0.3304,Y -4.738,Z 38,A -2.904,B 0,C 0,E1 0.1598,E2 90.0716} C_DIS
LIN {X -0.3304,Y -4.738,Z 38,A -2.904,B 0,C 0,E1 0.1598,E2 90.0716} C_DIS
Enddeposition()
LIN {X 0.0317,Y -5.6871,Z 38,A -2.9301,B 0,C 0,E1 0.1598,E2 90.0705} C_DIS
Startdeposition()
$VEL.CP = VEL_PRINT
LIN {X -0.8105,Y -5.6265,Z 38,A -2.9595,B 0,C 0,E1 0.1598,E2 90.0716} C_DIS
LIN {X -1.905,Y -5.3613,Z 38,A -2.9884,B 0,C 0,E1 0.1598,E2 90.0716} C_DIS
LIN {X -2.702,Y -5.002,Z 38,A -3.0024,B 0,C 0,E1 0.1598,E2 90.0716} C_DIS
LIN {X -3.273,Y -4.6537,Z 38,A -3.0086,B 0,C 0,E1 0.1598,E2 90.0716} C_DIS
LIN {X -3.8784,Y -4.1568,Z 38,A -3.0096,B 0,C 0,E1 0.1598,E2 90.0714} C_DIS
LIN {X -4.4478,Y -3.5405,Z 38,A -3.0043,B 0,C 0,E1 0.1598,E2 90.0714} C_DIS
LIN {X -4.9209,Y -2.8475,Z 38,A -2.9923,B 0,C 0,E1 0.1598,E2 90.0714} C_DIS
LIN {X -5.2864,Y -2.0922,Z 38,A -2.9737,B 0,C 0,E1 0.1598,E2 90.0713} C_DIS
LIN {X -5.5351,Y -1.2909,Z 38,A -2.9488,B 0,C 0,E1 0.1598,E2 90.0713} C_DIS
LIN {X -5.6664,Y -0.4623,Z 38,A -2.9186,B 0,C 0,E1 0.1598,E2 90.0713} C_DIS
LIN {X -5.6874,Y 0.1671,Z 38,A -2.8929,B 0,C 0,E1 0.1598,E2 90.0715} C_DIS
LIN {X -5.4354,Y 1.681,Z 38,A -2.8186,B 0,C 0,E1 0.1598,E2 90.0707} C_DIS
LIN {X -5.0228,Y 2.6646,Z 38,A -2.7623,B 0,C 0,E1 0.1598,E2 90.0713} C_DIS
LIN {X -4.6261,Y 3.3017,Z 38,A -2.7211,B 0,C 0,E1 0.1598,E2 90.0717} C_DIS
LIN {X -4.1509,Y 3.8821,Z 38,A -2.6791,B 0,C 0,E1 0.1598,E2 90.0718} C_DIS
LIN {X -3.4598,Y 4.5163,Z 38,A -2.6267,B 0,C 0,E1 0.1598,E2 90.0718} C_DIS
LIN {X -2.0797,Y 5.2971,Z 38,A -2.5427,B 0,C 0,E1 0.1598,E2 90.0719} C_DIS
LIN {X -1.2291,Y 5.5499,Z 38,A -2.5009,B 0,C 0,E1 0.1598,E2 90.0722} C_DIS
LIN {X -0.528,Y 5.6607,Z 38,A -2.4703,B 0,C 0,E1 0.1598,E2 90.0722} C_DIS
LIN {X 0.1815,Y 5.6813,Z 38,A -2.4433,B 0,C 0,E1 0.1598,E2 90.0723} C_DIS
LIN {X 1.0642,Y 5.5901,Z 38,A -2.4146,B 0,C 0,E1 0.1598,E2 90.0723} C_DIS
LIN {X 2.1412,Y 5.2671,Z 38,A -2.3885,B 0,C 0,E1 0.1598,E2 90.0723} C_DIS
LIN {X 2.8867,Y 4.8957,Z 38,A -2.3768,B 0,C 0,E1 0.1598,E2 90.0723} C_DIS
LIN {X 3.5719,Y 4.4221,Z 38,A -2.3716,B 0,C 0,E1 0.1598,E2 90.0723} C_DIS
LIN {X 4.1802,Y 3.853,Z 38,A -2.3733,B 0,C 0,E1 0.1598,E2 90.0723} C_DIS
LIN {X 4.6991,Y 3.2014,Z 38,A -2.3819,B 0,C 0,E1 0.1598,E2 90.0721} C_DIS
LIN {X 5.115,Y 2.4795,Z 38,A -2.3972,B 0,C 0,E1 0.1598,E2 90.0721} C_DIS
LIN {X 5.4229,Y 1.7055,Z 38,A -2.4188,B 0,C 0,E1 0.1598,E2 90.072} C_DIS
LIN {X 5.6142,Y 0.8949,Z 38,A -2.4462,B 0,C 0,E1 0.1598,E2 90.072} C_DIS
LIN {X 5.6847,Y 0.0649,Z 38,A -2.479,B 0,C 0,E1 0.1598,E2 90.0719} C_DIS
LIN {X 5.6339,Y -0.7666,Z 38,A -2.5162,B 0,C 0,E1 0.1598,E2 90.0719} C_DIS
LIN {X 5.4603,Y -1.5815,Z 38,A -2.5574,B 0,C 0,E1 0.1598,E2 90.0718} C_DIS
LIN {X 5.1684,Y -2.3615,Z 38,A -2.6014,B 0,C 0,E1 0.1598,E2 90.0718} C_DIS
LIN {X 4.768,Y -3.0916,Z 38,A -2.6472,B 0,C 0,E1 0.1598,E2 90.0718} C_DIS
LIN {X 4.2647,Y -3.7549,Z 38,A -2.694,B 0,C 0,E1 0.1598,E2 90.0718} C_DIS
LIN {X 3.6705,Y -4.3382,Z 38,A -2.7407,B 0,C 0,E1 0.1598,E2 90.0718} C_DIS
LIN {X 2.997,Y -4.8279,Z 38,A -2.7863,B 0,C 0,E1 0.1598,E2 90.0718} C_DIS
LIN {X 2.2598,Y -5.2151,Z 38,A -2.8299,B 0,C 0,E1 0.1598,E2 90.0718} C_DIS
LIN {X 1.4734,Y -5.489,Z 38,A -2.8705,B 0,C 0,E1 0.1598,E2 90.0718} C_DIS
LIN {X 0.6554,Y -5.646,Z 38,A -2.9072,B 0,C 0,E1 0.1598,E2 90.0717} C_DIS
LIN {X 0.0317,Y -5.6871,Z 38,A -2.9318,B 0,C 0,E1 0.1598,E2 90.0717} C_DIS
Enddeposition()
LIN {X 0.0317,Y -5.6871,Z 38,A -2.9318,B 0,C 0,E1 0.1598,E2 90.0717} C_DIS
Startdeposition()
$VEL.CP = VEL_PRINT
LIN {X 0.5776,Y -6.5946,Z 38,A -2.95,B 0,C 0,E1 0.1598,E2 90.0711} C_DIS
LIN {X 1.6078,Y -6.4253,Z 38,A -2.9055,B 0,C 0,E1 0.1598,E2 90.0717} C_DIS
LIN {X 2.487,Y -6.1336,Z 38,A -2.8609,B 0,C 0,E1 0.1598,E2 90.0717} C_DIS
LIN {X 3.1568,Y -5.817,Z 38,A -2.8228,B 0,C 0,E1 0.1598,E2 90.0717} C_DIS
LIN {X 3.7874,Y -5.4278,Z 38,A -2.7831,B 0,C 0,E1 0.1598,E2 90.0717} C_DIS
LIN {X 4.3701,Y -4.9701,Z 38,A -2.7421,B 0,C 0,E1 0.1598,E2 90.0718} C_DIS
LIN {X 4.8987,Y -4.4508,Z 38,A -2.7006,B 0,C 0,E1 0.1598,E2 90.0718} C_DIS
LIN {X 5.3651,Y -3.8753,Z 38,A -2.6589,B 0,C 0,E1 0.1598,E2 90.0718} C_DIS
LIN {X 5.7648,Y -3.2514,Z 38,A -2.6176,B 0,C 0,E1 0.1598,E2 90.0718} C_DIS
LIN {X 6.0925,Y -2.5868,Z 38,A -2.5772,B 0,C 0,E1 0.1598,E2 90.0718} C_DIS
LIN {X 6.3445,Y -1.89,Z 38,A -2.5382,B 0,C 0,E1 0.1598,E2 90.0719} C_DIS
LIN {X 6.5147,Y -1.1688,Z 38,A -2.5011,B 0,C 0,E1 0.1598,E2 90.0719} C_DIS
LIN {X 6.6045,Y -0.4333,Z 38,A -2.4665,B 0,C 0,E1 0.1598,E2 90.0719} C_DIS
LIN {X 6.6102,Y 0.3076,Z 38,A -2.4347,B 0,C 0,E1 0.1598,E2 90.072} C_DIS
LIN {X 6.5358,Y 1.0448,Z 38,A -2.406,B 0,C 0,E1 0.1598,E2 90.072} C_DIS
LIN {X 6.3782,Y 1.7689,Z 38,A -2.381,B 0,C 0,E1 0.1598,E2 90.072} C_DIS
LIN {X 6.1412,Y 2.471,Z 38,A -2.3598,B 0,C 0,E1 0.1598,E2 90.0721} C_DIS
LIN {X 5.828,Y 3.1425,Z 38,A -2.3428,B 0,C 0,E1 0.1598,E2 90.0721} C_DIS
LIN {X 5.4398,Y 3.7736,Z 38,A -2.3302,B 0,C 0,E1 0.1598,E2 90.0722} C_DIS
LIN {X 4.9833,Y 4.3576,Z 38,A -2.3222,B 0,C 0,E1 0.1598,E2 90.0722} C_DIS
LIN {X 4.4648,Y 4.8872,Z 38,A -2.3189,B 0,C 0,E1 0.1598,E2 90.0723} C_DIS
LIN {X 3.8904,Y 5.3554,Z 38,A -2.3202,B 0,C 0,E1 0.1598,E2 90.0723} C_DIS
LIN {X 3.2667,Y 5.7554,Z 38,A -2.3262,B 0,C 0,E1 0.1598,E2 90.0723} C_DIS
LIN {X 2.6039,Y 6.0865,Z 38,A -2.3366,B 0,C 0,E1 0.1598,E2 90.0723} C_DIS
LIN {X 1.9074,Y 6.3396,Z 38,A -2.3516,B 0,C 0,E1 0.1598,E2 90.0723} C_DIS
LIN {X 1.0044,Y 6.5468,Z 38,A -2.3761,B 0,C 0,E1 0.1598,E2 90.0723} C_DIS
LIN {X -0.0177,Y 6.6182,Z 38,A -2.4108,B 0,C 0,E1 0.1598,E2 90.0723} C_DIS
LIN {X -0.7121,Y 6.5801,Z 38,A -2.4381,B 0,C 0,E1 0.1598,E2 90.0723} C_DIS
LIN {X -1.399,Y 6.47,Z 38,A -2.4681,B 0,C 0,E1 0.1598,E2 90.0723} C_DIS
LIN {X -2.0704,Y 6.2883,Z 38,A -2.5005,B 0,C 0,E1 0.1598,E2 90.0723} C_DIS
LIN {X -2.7188,Y 6.0362,Z 38,A -2.5351,B 0,C 0,E1 0.1598,E2 90.0722} C_DIS
LIN {X -3.3369,Y 5.7169,Z 38,A -2.5714,B 0,C 0,E1 0.1598,E2 90.0721} C_DIS
LIN {X -3.9182,Y 5.3349,Z 38,A -2.609,B 0,C 0,E1 0.1598,E2 90.0721} C_DIS
LIN {X -4.4563,Y 4.8942,Z 38,A -2.6474,B 0,C 0,E1 0.1598,E2 90.0719} C_DIS
LIN {X -4.945,Y 4.3993,Z 38,A -2.6864,B 0,C 0,E1 0.1598,E2 90.0719} C_DIS
LIN {X -5.3799,Y 3.8564,Z 38,A -2.7253,B 0,C 0,E1 0.1598,E2 90.0718} C_DIS
LIN {X -5.7546,Y 3.2704,Z 38,A -2.7639,B 0,C 0,E1 0.1598,E2 90.0718} C_DIS
LIN {X -6.066,Y 2.6484,Z 38,A -2.8016,B 0,C 0,E1 0.1598,E2 90.0716} C_DIS
LIN {X -6.3135,Y 1.9983,Z 38,A -2.8382,B 0,C 0,E1 0.1598,E2 90.0716} C_DIS
LIN {X -6.4881,Y 1.3249,Z 38,A -2.8731,B 0,C 0,E1 0.1598,E2 90.0716} C_DIS
LIN {X -6.5896,Y 0.6367,Z 38,A -2.9059,B 0,C 0,E1 0.1598,E2 90.0715} C_DIS
LIN {X -6.6119,Y -0.3923,Z 38,A -2.95,B 0,C 0,E1 0.1598,E2 90.0711} C_DIS
LIN {X -6.4972,Y -1.272,Z 38,A -2.9831,B 0,C 0,E1 0.1598,E2 90.0712} C_DIS
LIN {X -6.3254,Y -1.9606,Z 38,A -3.0061,B 0,C 0,E1 0.1598,E2 90.0713} C_DIS
LIN {X -6.0787,Y -2.626,Z 38,A -3.0252,B 0,C 0,E1 0.1598,E2 90.0713} C_DIS
LIN {X -5.7616,Y -3.261,Z 38,A -3.0405,B 0,C 0,E1 0.1598,E2 90.0713} C_DIS
LIN {X -5.3794,Y -3.859,Z 38,A -3.0518,B 0,C 0,E1 0.1598,E2 90.0713} C_DIS
LIN {X -4.9353,Y -4.4128,Z 38,A -3.059,B 0,C 0,E1 0.1598,E2 90.0713} C_DIS
LIN {X -4.4336,Y -4.9146,Z 38,A -3.0619,B 0,C 0,E1 0.1598,E2 90.0713} C_DIS
LIN {X -3.8821,Y -5.3613,Z 38,A -3.0606,B 0,C 0,E1 0.1598,E2 90.0713} C_DIS
LIN {X -3.1324,Y -5.8357,Z 38,A -3.0532,B 0,C 0,E1 0.1598,E2 90.0713} C_DIS
LIN {X -2.1896,Y -6.2485,Z 38,A -3.0362,B 0,C 0,E1 0.1598,E2 90.0714} C_DIS
LIN {X -1.5188,Y -6.4428,Z 38,A -3.0199,B 0,C 0,E1 0.1598,E2 90.0715} C_DIS
LIN {X -0.8316,Y -6.5672,Z 38,A -3,B 0,C 0,E1 0.1598,E2 90.0715} C_DIS
LIN {X 0.0397,Y -6.6206,Z 38,A -2.9703,B 0,C 0,E1 0.1598,E2 90.0716} C_DIS
Enddeposition()
LIN {X 0.0397,Y -6.6206,Z 38,A -2.9703,B 0,C 0,E1 0.1598,E2 90.0716} C_DIS
Startdeposition()
$VEL.CP = VEL_PRINT
LIN {X -0.2474,Y -7.5533,Z 38,A -3.0201,B 0,C 0,E1 0.1598,E2 90.071} C_DIS
LIN {X -1.3339,Y -7.4394,Z 38,A -3.0556,B 0,C 0,E1 0.1598,E2 90.0715} C_DIS
LIN {X -2.4146,Y -7.1574,Z 38,A -3.0833,B 0,C 0,E1 0.1598,E2 90.0715} C_DIS
LIN {X -3.3195,Y -6.7884,Z 38,A -3.1007,B 0,C 0,E1 0.1598,E2 90.0713} C_DIS
LIN {X -4.3117,Y -6.2011,Z 38,A -3.1121,B 0,C 0,E1 0.1598,E2 90.0713} C_DIS
LIN {X -4.9739,Y -5.6816,Z 38,A -3.1144,B 0,C 0,E1 0.1598,E2 90.0713} C_DIS
LIN {X -5.5764,Y -5.094,Z 38,A -3.1116,B 0,C 0,E1 0.1598,E2 90.0713} C_DIS
LIN {X -6.1087,Y -4.4421,Z 38,A -3.1034,B 0,C 0,E1 0.1598,E2 90.0713} C_DIS
LIN {X -6.5644,Y -3.7344,Z 38,A -3.0902,B 0,C 0,E1 0.1598,E2 90.0712} C_DIS
LIN {X -7.0254,Y -2.7887,Z 38,A -3.0668,B 0,C 0,E1 0.1598,E2 90.0709} C_DIS
LIN {X -7.3453,Y -1.7795,Z 38,A -3.0358,B 0,C 0,E1 0.1598,E2 90.071} C_DIS
LIN {X -7.5178,Y -0.7716,Z 38,A -2.9995,B 0,C 0,E1 0.1598,E2 90.071} C_DIS
LIN {X -7.551,Y 0.3132,Z 38,A -2.9547,B 0,C 0,E1 0.1598,E2 90.071} C_DIS
LIN {X -7.4668,Y 1.1634,Z 38,A -2.916,B 0,C 0,E1 0.1598,E2 90.0713} C_DIS
LIN {X -7.2211,Y 2.227,Z 38,A -2.8618,B 0,C 0,E1 0.1598,E2 90.0712} C_DIS
LIN {X -6.9114,Y 3.0572,Z 38,A -2.8154,B 0,C 0,E1 0.1598,E2 90.0713} C_DIS
LIN {X -6.2243,Y 4.2835,Z 38,A -2.738,B 0,C 0,E1 0.1598,E2 90.0713} C_DIS
LIN {X -5.787,Y 4.8595,Z 38,A -2.6979,B 0,C 0,E1 0.1598,E2 90.0717} C_DIS
LIN {X -5.0327,Y 5.6388,Z 38,A -2.6371,B 0,C 0,E1 0.1598,E2 90.0717} C_DIS
LIN {X -4.2503,Y 6.2433,Z 38,A -2.5829,B 0,C 0,E1 0.1598,E2 90.072} C_DIS
LIN {X -3.5741,Y 6.6536,Z 38,A -2.5406,B 0,C 0,E1 0.1598,E2 90.072} C_DIS
LIN {X -2.4411,Y 7.153,Z 38,A -2.4777,B 0,C 0,E1 0.1598,E2 90.0722} C_DIS
LIN {X -1.0929,Y 7.4781,Z 38,A -2.4142,B 0,C 0,E1 0.1598,E2 90.0723} C_DIS
LIN {X -0.0881,Y 7.5533,Z 38,A -2.374,B 0,C 0,E1 0.1598,E2 90.0724} C_DIS
LIN {X 0.9182,Y 7.5011,Z 38,A -2.3391,B 0,C 0,E1 0.1598,E2 90.0724} C_DIS
LIN {X 1.9279,Y 7.3067,Z 38,A -2.31,B 0,C 0,E1 0.1598,E2 90.0724} C_DIS
LIN {X 2.7492,Y 7.0404,Z 38,A -2.291,B 0,C 0,E1 0.1598,E2 90.0724} C_DIS
LIN {X 3.764,Y 6.548,Z 38,A -2.2743,B 0,C 0,E1 0.1598,E2 90.0724} C_DIS
LIN {X 4.454,Y 6.0998,Z 38,A -2.268,B 0,C 0,E1 0.1598,E2 90.0724} C_DIS
LIN {X 5.3208,Y 5.3679,Z 38,A -2.2669,B 0,C 0,E1 0.1598,E2 90.0722} C_DIS
LIN {X 6.2086,Y 4.3073,Z 38,A -2.2789,B 0,C 0,E1 0.1598,E2 90.0718} C_DIS
Enddeposition()
END
